(* POU TN_INPUT_CONTROL, ST *)
FUNCTION_BLOCK TN_INPUT_CONTROL
VAR_IN_OUT
	Xus_TN_SCREEN : us_TN_SCREEN;
	Xus_TN_INPUT_CONTROL : us_TN_INPUT_CONTROL;
END_VAR
VAR
	FB_TN_INPUT_SELECT_POPUP : TN_INPUT_SELECT_POPUP;
	FB_TN_INPUT_SELECT_TEXT : TN_INPUT_SELECT_TEXT;
	FB_TN_SC_WRITE_C : TN_SC_WRITE_C;
	FB_TN_INPUT_EDIT_LINE : TN_INPUT_EDIT_LINE;
END_VAR
VAR
	in_index : INT;
	in_Scroll_Offset : INT;
	in_Focus_new : INT;
	in_Focus_alt : INT;
	bo_Tool_Tip_Update : BOOL;
END_VAR

(*
version 1.0		10. mai 2010
programmer		ks
tested by		ks

TN_INPUT_CONTROL dient zur verwaltung und grafischen Darstellung der INPUT_CONTROL Elemente
*)
(* Bearbeitung freigegeben ? *)
IF (Xus_TN_INPUT_CONTROL.bo_Enable = FALSE) OR (Xus_TN_SCREEN.bo_Menue_Bar_Dialog = TRUE) THEN
	RETURN;
END_IF;

(* Fokus Reset durchführen *)
IF (Xus_TN_INPUT_CONTROL.bo_Reset_Fokus = TRUE) THEN
	Xus_TN_INPUT_CONTROL.bo_Reset_Fokus := FALSE;

	FOR in_index := INT#01 TO Xus_TN_INPUT_CONTROL.in_Count DO
		Xus_TN_INPUT_CONTROL.usa_TN_INPUT_CONTROL_DATA[in_index].bo_Focus := FALSE;
	END_FOR;

	IF (Xus_TN_INPUT_CONTROL.in_Count >= INT#01) THEN
		Xus_TN_INPUT_CONTROL.usa_TN_INPUT_CONTROL_DATA[1].bo_Focus := TRUE;
		Xus_TN_INPUT_CONTROL.in_Focus_at := INT#01;
	END_IF;

	Xus_TN_INPUT_CONTROL.bo_Update_all := TRUE;
END_IF;

IF (Xus_TN_SCREEN.bo_Modal_Dialog = FALSE) THEN
	(* TAB-Taste für Control-element wechsel auswerten *)
	IF (Xus_TN_SCREEN.by_Input_Exten_Code = BYTE#09) THEN

		in_Scroll_Offset := INT#01;

		(* Cursor-Oben Taste *)
	ELSIF (Xus_TN_SCREEN.by_Input_Exten_Code = BYTE#65) THEN

		in_Scroll_Offset := -1;

		(* Cursor-unten Taste *)
	ELSIF (Xus_TN_SCREEN.by_Input_Exten_Code = BYTE#66) THEN

		in_Scroll_Offset := INT#01;

	END_IF;
END_IF;

IF (in_Scroll_Offset <> INT#00) THEN  
	(* Grenzwerte überprüfen                                            *)

	Xus_TN_INPUT_CONTROL.in_Focus_at:=LIMIT(INT#01,Xus_TN_INPUT_CONTROL.in_Focus_at,Xus_TN_INPUT_CONTROL.in_Count);

	in_Focus_new := Xus_TN_INPUT_CONTROL.in_Focus_at + in_Scroll_Offset;

	IF (in_Focus_new > Xus_TN_INPUT_CONTROL.in_Count) THEN
		in_Focus_new := INT#1;
	END_IF;

	IF (in_Focus_new < INT#01) THEN
		in_Focus_new := Xus_TN_INPUT_CONTROL.in_Count;
	END_IF;

	in_Focus_alt := Xus_TN_INPUT_CONTROL.in_Focus_at;

	(* aktuellen Element den Fokus entziehen *)
	Xus_TN_INPUT_CONTROL.usa_TN_INPUT_CONTROL_DATA[in_Focus_alt].bo_Focus := FALSE;
	Xus_TN_INPUT_CONTROL.usa_TN_INPUT_CONTROL_DATA[in_Focus_alt].bo_Update_Input := TRUE;

	(* neuem Element den Fokus geben *)
	Xus_TN_INPUT_CONTROL.usa_TN_INPUT_CONTROL_DATA[in_Focus_new].bo_Focus  := TRUE;
	Xus_TN_INPUT_CONTROL.usa_TN_INPUT_CONTROL_DATA[in_Focus_new].bo_Update_Input := TRUE;

	Xus_TN_INPUT_CONTROL.in_Focus_at := in_Focus_new;

	bo_Tool_Tip_Update := TRUE;
	in_Scroll_Offset := INT#00;

END_IF;

(* Alle Elemente updaten ? *)
IF (Xus_TN_INPUT_CONTROL.bo_Update_all = TRUE) THEN
	FOR in_index := 1 TO Xus_TN_INPUT_CONTROL.in_Count DO
		Xus_TN_INPUT_CONTROL.usa_TN_INPUT_CONTROL_DATA[in_index].bo_Update_All := TRUE;
	END_FOR;
	Xus_TN_INPUT_CONTROL.bo_Update_all := FALSE;
	bo_Tool_Tip_Update := TRUE;
END_IF;

FOR in_index := 1 TO Xus_TN_INPUT_CONTROL.in_Count DO

	IF (Xus_TN_INPUT_CONTROL.usa_TN_INPUT_CONTROL_DATA[in_index].in_Type > INT#00) THEN

		IF (Xus_TN_INPUT_CONTROL.usa_TN_INPUT_CONTROL_DATA[in_index].bo_Focus = TRUE) THEN

			Xus_TN_INPUT_CONTROL.usa_TN_INPUT_CONTROL_DATA[in_index].by_Input_ASCII_Code  := Xus_TN_SCREEN.by_Input_ASCII_Code;
			Xus_TN_INPUT_CONTROL.usa_TN_INPUT_CONTROL_DATA[in_index].by_Input_Exten_Code  := Xus_TN_SCREEN.by_Input_Exten_Code;
			Xus_TN_INPUT_CONTROL.usa_TN_INPUT_CONTROL_DATA[in_index].bo_Input_ASCII_IsNum := Xus_TN_SCREEN.bo_Input_ASCII_IsNum;

			(* Tool-Tip Text ausgeben *)
			IF (bo_Tool_Tip_Update = TRUE) THEN

				FB_TN_SC_WRITE_C(	Iin_Y := Xus_TN_INPUT_CONTROL.in_ToolTip_Y,
									Iin_X := Xus_TN_INPUT_CONTROL.in_ToolTip_X,
									Iby_ATTR := Xus_TN_INPUT_CONTROL.by_ToolTip_Attr,
									Iin_OPTION := INT#02, (* Center-String *)
									Iin_LENGTH := Xus_TN_INPUT_CONTROL.in_ToolTip_Size,
									Ist_STRING := Xus_TN_INPUT_CONTROL.usa_TN_INPUT_CONTROL_DATA[in_index].st_Input_ToolTip,
									Xus_TN_SCREEN := Xus_TN_SCREEN);

				(* Flag rücksetzen *)
				bo_Tool_Tip_Update := FALSE;
			END_IF;
		END_IF;

		CASE Xus_TN_INPUT_CONTROL.usa_TN_INPUT_CONTROL_DATA[in_index].in_Type OF
		1:
			(* Edit-Line bearbeiten *)
			FB_TN_INPUT_EDIT_LINE(	Xus_TN_INPUT_CONTROL_DATA := Xus_TN_INPUT_CONTROL.usa_TN_INPUT_CONTROL_DATA[in_index],
									Xus_TN_SCREEN := Xus_TN_SCREEN);
		2:
			(* Select-Text bearbeiten *)
			FB_TN_INPUT_SELECT_TEXT(	Xus_TN_INPUT_CONTROL_DATA := Xus_TN_INPUT_CONTROL.usa_TN_INPUT_CONTROL_DATA[in_index],
										Xus_TN_SCREEN := Xus_TN_SCREEN);
		3:
			(* Select-Popup bearbeiten *)
			FB_TN_INPUT_SELECT_POPUP(	Xus_TN_INPUT_CONTROL_DATA := Xus_TN_INPUT_CONTROL.usa_TN_INPUT_CONTROL_DATA[in_index],
										Xus_TN_SCREEN := Xus_TN_SCREEN);
		END_CASE;

		IF (Xus_TN_INPUT_CONTROL.usa_TN_INPUT_CONTROL_DATA[in_index].bo_Focus = TRUE) THEN

			(* Cursor position von Element auf Screen übertragen *)
			Xus_TN_SCREEN.in_Cursor_X := Xus_TN_INPUT_CONTROL.usa_TN_INPUT_CONTROL_DATA[in_index].in_Cursor_X;
			Xus_TN_SCREEN.in_Cursor_Y := Xus_TN_INPUT_CONTROL.usa_TN_INPUT_CONTROL_DATA[in_index].in_Cursor_Y;

		END_IF;
	END_IF;
END_FOR;

(* revision history
ks	10. mai. 2010	rev 1.0
	original version
*)
END_FUNCTION_BLOCK

(* POU TN_INPUT_SELECT_POPUP, ST *)
FUNCTION_BLOCK TN_INPUT_SELECT_POPUP
VAR
	in_index : INT;
	in_Element_Count : INT;
	by_Cur_Key : BYTE;
	by_Attr : BYTE;
	st_String : STRING;
END_VAR
VAR
	us_TN_MENU_POPUP : us_TN_MENU_POPUP;
	FB_TN_INPUT_MENU_POPUP : TN_INPUT_MENU_POPUP;
	FB_TN_SC_WRITE : TN_SC_WRITE;
END_VAR
VAR_IN_OUT
	Xus_TN_SCREEN : us_TN_SCREEN;
	Xus_TN_INPUT_CONTROL_DATA : us_TN_INPUT_CONTROL_DATA;
END_VAR

(*
version 1.1		06. apr 2011
programmer		ks
tested by			ks

TN_SELECT_POPUP dient zur verwaltung und darstellung eines POPUP-Dialogs zur Elementeauswahl
*)
(* Benutzereingabe auswerten -> Selektion Text n *)
IF (Xus_TN_INPUT_CONTROL_DATA.bo_Focus = TRUE) THEN

	by_Cur_Key := Xus_TN_INPUT_CONTROL_DATA.by_Input_Exten_Code;

	IF (us_TN_MENU_POPUP.bo_Activ = FALSE) THEN
		us_TN_MENU_POPUP.by_Input_Exten_Code := BYTE#00;

		(* Return-Taste auswerten *)
		IF (by_Cur_Key = BYTE#13) THEN
			(* Popup-Menu parameter übergeben *)
			us_TN_MENU_POPUP.in_Y := Xus_TN_INPUT_CONTROL_DATA.in_Y;
			us_TN_MENU_POPUP.in_X := Xus_TN_INPUT_CONTROL_DATA.in_X;
			us_TN_MENU_POPUP.by_Attr_mF := Xus_TN_INPUT_CONTROL_DATA.by_Attr_mF;
			us_TN_MENU_POPUP.by_Attr_oF := Xus_TN_INPUT_CONTROL_DATA.by_Attr_oF;
			us_TN_MENU_POPUP.st_Menu_Text := Xus_TN_INPUT_CONTROL_DATA.st_Input_Data;
			us_TN_MENU_POPUP.bo_Create := TRUE;
			us_TN_MENU_POPUP.in_Cur_Item := INT#00;
		END_IF;

		IF (us_TN_MENU_POPUP.in_Cur_Item > INT#00) THEN
			Xus_TN_INPUT_CONTROL_DATA.in_selected := us_TN_MENU_POPUP.in_Cur_Item;
			Xus_TN_INPUT_CONTROL_DATA.bo_Input_Entered := TRUE;
			Xus_TN_INPUT_CONTROL_DATA.bo_Update_Input := TRUE;
			us_TN_MENU_POPUP.in_Cur_Item := INT#00;
		END_IF;

	ELSE
		us_TN_MENU_POPUP.by_Input_Exten_Code := by_Cur_Key;
	END_IF;

	(* Popup-Menu zyklisch aufrufen *)
	FB_TN_INPUT_MENU_POPUP(Xus_TN_MENU_POPUP := us_TN_MENU_POPUP, Xus_TN_SCREEN := Xus_TN_SCREEN);

END_IF;

(* Aktualisierung der Anzeige *)
IF (Xus_TN_INPUT_CONTROL_DATA.bo_Update_Input = TRUE) OR (Xus_TN_INPUT_CONTROL_DATA.bo_Update_All = TRUE) THEN

	(* Title-Text ausgeben *)
	IF Xus_TN_INPUT_CONTROL_DATA.bo_Update_All = TRUE THEN

		IF (Xus_TN_INPUT_CONTROL_DATA.in_Title_X_Offset = INT#00) AND (Xus_TN_INPUT_CONTROL_DATA.in_Title_Y_Offset = INT#00) THEN
			(* wenn Offset X,Y =0 dann Titlestring links vom Element positionieren *)
			FB_TN_SC_WRITE.Iin_Y := Xus_TN_INPUT_CONTROL_DATA.in_Y;
			FB_TN_SC_WRITE.Iin_X := Xus_TN_INPUT_CONTROL_DATA.in_X - LEN(Xus_TN_INPUT_CONTROL_DATA.st_Title_String);

		ELSE
			(* Title-Text durch Row, Color-Offset ausgeben *)
			FB_TN_SC_WRITE.Iin_Y := Xus_TN_INPUT_CONTROL_DATA.in_Y + Xus_TN_INPUT_CONTROL_DATA.in_Title_Y_Offset;
			FB_TN_SC_WRITE.Iin_X := Xus_TN_INPUT_CONTROL_DATA.in_X + Xus_TN_INPUT_CONTROL_DATA.in_Title_X_Offset;
		END_IF;

		(* Title-Text durch Row, Color-Offset ausgeben *)
		FB_TN_SC_WRITE(	Iby_ATTR := Xus_TN_INPUT_CONTROL_DATA.by_Title_Attr,
						Ist_STRING := Xus_TN_INPUT_CONTROL_DATA.st_Title_String,
						Xus_TN_SCREEN := Xus_TN_SCREEN);
	END_IF;

	in_Element_Count := ELEMENT_COUNT(SEP:=BYTE#35,ELEMENT:=Xus_TN_INPUT_CONTROL_DATA.st_Input_Data);

	IF in_Element_Count > INT#00 THEN

		Xus_TN_INPUT_CONTROL_DATA.in_selected:=LIMIT(1,Xus_TN_INPUT_CONTROL_DATA.in_selected,in_Element_Count);

		in_index := Xus_TN_INPUT_CONTROL_DATA.in_selected;

		st_String := ELEMENT_GET(SEP:=BYTE#35,POS:=in_index - 1,ELEMENT:=Xus_TN_INPUT_CONTROL_DATA.st_Input_Data);

		st_String:= FIX(str:=st_String,
						L:=LEN(Xus_TN_INPUT_CONTROL_DATA.st_Input_Mask),
						C:=BYTE#32,
						M:=Xus_TN_INPUT_CONTROL_DATA.in_Input_Option);


		Xus_TN_INPUT_CONTROL_DATA.st_Input_String := st_String;

		IF Xus_TN_INPUT_CONTROL_DATA.bo_Focus = TRUE THEN
			by_Attr := Xus_TN_INPUT_CONTROL_DATA.by_Attr_mF;
		ELSE
			by_Attr := Xus_TN_INPUT_CONTROL_DATA.by_Attr_oF;
		END_IF;

		FB_TN_SC_WRITE(	Iin_X := Xus_TN_INPUT_CONTROL_DATA.in_X,
								Iin_Y := Xus_TN_INPUT_CONTROL_DATA.in_Y,
								Iby_ATTR := by_Attr,
								Ist_STRING := st_String,
								Xus_TN_SCREEN := Xus_TN_SCREEN );
	END_IF;

	(* Cursor auf aktuelle Position setzen *)
	Xus_TN_INPUT_CONTROL_DATA.in_Cursor_X := Xus_TN_INPUT_CONTROL_DATA.in_X;
	Xus_TN_INPUT_CONTROL_DATA.in_Cursor_Y := Xus_TN_INPUT_CONTROL_DATA.in_Y;

	(* Update-Flag's rücksetzen *)
	Xus_TN_INPUT_CONTROL_DATA.bo_Update_All   := FALSE;
	Xus_TN_INPUT_CONTROL_DATA.bo_Update_Input := FALSE;

END_IF;

(* revision history

ks	06. apr. 2011	rev 1.1
	list_len und list_get durch element_count und element_get ersetzt

ks	10. mai. 2010	rev 1.0
	original version
*)
END_FUNCTION_BLOCK

(* POU TN_INPUT_MENU_POPUP, ST *)
FUNCTION_BLOCK TN_INPUT_MENU_POPUP
VAR
	FB_TN_SC_AREA_SAVE : TN_SC_AREA_SAVE;
	FB_TN_SC_AREA_RESTORE : TN_SC_AREA_RESTORE;
	FB_TN_SC_LINE : TN_SC_LINE;
	FB_TN_SC_ADD_SHADOW : TN_SC_ADD_SHADOW;
	FB_TN_SC_BOX : TN_SC_BOX;
	FB_TN_SC_WRITE_C : TN_SC_WRITE_C;
END_VAR
VAR
	in_ROW : INT;
	in_ROWS : INT;
	in_COL : INT;
	in_COLS : INT;
	in_index : INT;
	in_Count : INT;
	in_Scroll_Offset : INT;
	by_ATTR : BYTE;
END_VAR
VAR_IN_OUT
	Xus_TN_MENU_POPUP : us_TN_MENU_POPUP;
	Xus_TN_SCREEN : us_TN_SCREEN;
END_VAR

(*
version 1.1		06. apr 2011
programmer		ks
tested by			ks

TN_MENU_POPUP dient zur verwaltung und darstellung eines MENU-POPUP
*)
(* sicherstellen das rechteck immer innerhalb screen positioniert wird *)

IF (Xus_TN_MENU_POPUP.bo_Activ = FALSE) AND (Xus_TN_MENU_POPUP.bo_Create = TRUE) THEN
	Xus_TN_MENU_POPUP.bo_Activ := TRUE;
	Xus_TN_MENU_POPUP.bo_Create := FALSE;
	Xus_TN_MENU_POPUP.bo_Destroy := FALSE;
	Xus_TN_MENU_POPUP.bo_Update := TRUE;

  (* Sub-Menu-Texte *)

	Xus_TN_MENU_POPUP.in_Menu_E_Count := ELEMENT_COUNT(SEP:=BYTE#35,ELEMENT:=Xus_TN_MENU_POPUP.st_Menu_Text);

	(* Anzahl Zeilen (Sub-Menu-Texte) bestimmen *)
	Xus_TN_MENU_POPUP.in_Rows := Xus_TN_MENU_POPUP.in_Menu_E_Count;

	(* längsten Sub-Menu-Text suchen *)
	Xus_TN_MENU_POPUP.in_Cols := INT#00;

	FOR in_Count := INT#01 TO Xus_TN_MENU_POPUP.in_Rows DO;
		Xus_TN_MENU_POPUP.in_Cols:=MAX(LEN(ELEMENT_GET(SEP:=BYTE#35,POS:=in_Count - 1,ELEMENT:=Xus_TN_MENU_POPUP.st_Menu_Text)),Xus_TN_MENU_POPUP.in_Cols);
	END_FOR;

	(* Horizontale Position überprüfen und korrigieren *)
	IF (Xus_TN_MENU_POPUP.in_X + Xus_TN_MENU_POPUP.in_Cols) > INT#75 THEN
		Xus_TN_MENU_POPUP.in_X := INT#79 - Xus_TN_MENU_POPUP.in_Cols - INT#04;
	END_IF;

  (* Vertikale Position überprüfen und korrigieren *)
	IF (Xus_TN_MENU_POPUP.in_Y + Xus_TN_MENU_POPUP.in_ROWS) > INT#21 THEN
		Xus_TN_MENU_POPUP.in_Y := INT#23 - Xus_TN_MENU_POPUP.in_ROWS - INT#2;
	END_IF;

	Xus_TN_SCREEN.bo_Modal_Dialog := TRUE;

	(* Hintergrund sichern *)
	FB_TN_SC_AREA_SAVE(	Iin_X1 := Xus_TN_MENU_POPUP.in_X,
									Iin_Y1 := Xus_TN_MENU_POPUP.in_Y,
									Iin_X2 := Xus_TN_MENU_POPUP.in_X + Xus_TN_MENU_POPUP.in_Cols + INT#04,
									Iin_Y2 := Xus_TN_MENU_POPUP.in_Y + Xus_TN_MENU_POPUP.in_Rows + INT#02,
									Xus_TN_SCREEN := Xus_TN_SCREEN);

	(* Rahmen für Submenu zeichnen *)
	FB_TN_SC_BOX(	Iin_X1 := Xus_TN_MENU_POPUP.in_X,
					Iin_Y1 := Xus_TN_MENU_POPUP.in_Y,
					Iin_X2 := Xus_TN_MENU_POPUP.in_X + Xus_TN_MENU_POPUP.in_Cols + INT#03,
					Iin_Y2 := Xus_TN_MENU_POPUP.in_Y + Xus_TN_MENU_POPUP.in_Rows + INT#01,
					Iby_FILL := BYTE#32, (* Füllung *)
					Iin_BORDER := INT#01, (* Single-Line Border *)
					Iby_ATTR := Xus_TN_MENU_POPUP.by_Attr_oF,
					Xus_TN_SCREEN := Xus_TN_SCREEN);

	(* Shadow für Submenu zeichnen *)
	FB_TN_SC_ADD_SHADOW(Iin_X1 := Xus_TN_MENU_POPUP.in_X + INT#1,
						Iin_Y1 := Xus_TN_MENU_POPUP.in_Y + INT#1,
						Iin_X2 := Xus_TN_MENU_POPUP.in_X + Xus_TN_MENU_POPUP.in_Cols + INT#04,
						Iin_Y2 := Xus_TN_MENU_POPUP.in_Y + Xus_TN_MENU_POPUP.in_Rows + INT#02,
						Iin_OPTION := INT#00,
						Xus_TN_SCREEN := Xus_TN_SCREEN);

	(* Parameter laden *)
	in_COL := Xus_TN_MENU_POPUP.in_X;
	in_ROW := Xus_TN_MENU_POPUP.in_Y;
	in_ROWS := Xus_TN_MENU_POPUP.in_Rows;
	in_COLS := Xus_TN_MENU_POPUP.in_Cols;

	(* Trennlinien zeichnen *)
	in_COLS := in_COLS + INT#02; (* Text um 2 Zeichen verlängern *)

	FOR in_Count := INT#01 TO Xus_TN_MENU_POPUP.in_Menu_E_Count DO;
		in_ROW := in_ROW + INT#01;

		IF ELEMENT_GET(SEP:=BYTE#35,POS:=in_Count - 1,ELEMENT:=Xus_TN_MENU_POPUP.st_Menu_Text) = '-' THEN

			FB_TN_SC_LINE(	Iin_Y1 := in_ROW,
							Iin_X1 := in_COL,
							Iin_Y2 := in_ROW,
							Iin_X2 := in_COL + in_COLS + INT#01,
							Iby_ATTR := Xus_TN_MENU_POPUP.by_Attr_oF,
							Iby_BORDER := BYTE#01,
							Xus_TN_SCREEN := Xus_TN_SCREEN);
		END_IF;
	END_FOR;
END_IF;

IF (Xus_TN_MENU_POPUP.bo_Activ = TRUE) THEN

	CASE BYTE_TO_INT(Xus_TN_MENU_POPUP.by_Input_Exten_Code) OF

	65: (* Cursor oben *)
		in_Scroll_Offset := -1;
		Xus_TN_MENU_POPUP.bo_Update := TRUE;

	66: (* Cursor unten *)
		in_Scroll_Offset := 1;
		Xus_TN_MENU_POPUP.bo_Update := TRUE;

	13:  (* Enter *)
		Xus_TN_MENU_POPUP.bo_Destroy := TRUE;

	27:  (* Escape*)
		Xus_TN_MENU_POPUP.bo_Destroy := TRUE;
		Xus_TN_MENU_POPUP.in_Cur_Item := INT#00;

	67..68: (* Cursor links oder rechts *)
		Xus_TN_MENU_POPUP.bo_Destroy := TRUE;
		Xus_TN_MENU_POPUP.in_Cur_Item := INT#00;

	END_CASE;
END_IF;

(* POPUP-Menu updaten *)
IF (Xus_TN_MENU_POPUP.bo_Activ = TRUE) AND (Xus_TN_MENU_POPUP.bo_Update = TRUE) THEN

	Xus_TN_MENU_POPUP.bo_Update := FALSE;

	(* überprüfung + nächstes anwählbares Sub-Menu suchen *)
	in_index := Xus_TN_MENU_POPUP.in_Cur_Item;

	IF (in_index < INT#01) OR (in_index > Xus_TN_MENU_POPUP.in_Menu_E_Count) THEN
		in_Scroll_Offset := INT#01;
		in_index := Xus_TN_MENU_POPUP.in_Menu_E_Count;
	END_IF;

	(* aktueller Index steht auf Trennzeichen -> ändern *)
	IF ELEMENT_GET(SEP:=BYTE#35,POS:=in_index-1,ELEMENT:=Xus_TN_MENU_POPUP.st_Menu_Text) = '-' THEN
		in_Scroll_Offset := INT#01;
	END_IF;

	(* Scroll-Offset *)
	IF in_Scroll_Offset <> INT#00 THEN

		FOR in_Count := INT#01 TO Xus_TN_MENU_POPUP.in_Menu_E_Count DO;

			in_index:=INC2(in_index,in_Scroll_Offset,1,Xus_TN_MENU_POPUP.in_Menu_E_Count);

			IF ELEMENT_GET(SEP:=BYTE#35,POS:=in_index - 1,ELEMENT:=Xus_TN_MENU_POPUP.st_Menu_Text) <> '-' THEN
				EXIT;
			END_IF;

		END_FOR;
	END_IF;

	Xus_TN_MENU_POPUP.in_Cur_Item := in_index;
	in_Scroll_Offset := INT#00;

	(* Parameter laden *)
	in_COL  := Xus_TN_MENU_POPUP.in_X;
	in_ROW  := Xus_TN_MENU_POPUP.in_Y;
	in_ROWS := Xus_TN_MENU_POPUP.in_Rows;
	in_COLS := Xus_TN_MENU_POPUP.in_Cols;

	(* SUB-MENU-Titel ausgeben *)
	in_COLS := in_COLS + INT#02; (* Text um 2 Zeichen verlängern *)

	FOR in_Count := INT#01 TO Xus_TN_MENU_POPUP.in_Menu_E_Count DO;

		in_ROW := in_ROW + INT#01;

		(* Zeichenfarbe bestimmen *)
		IF in_Count = Xus_TN_MENU_POPUP.in_Cur_Item THEN
			by_ATTR := Xus_TN_MENU_POPUP.by_Attr_mF;
		ELSE
			by_ATTR := Xus_TN_MENU_POPUP.by_Attr_oF;
		END_IF;

		FB_TN_SC_WRITE_C.Ist_STRING := ELEMENT_GET(SEP:=BYTE#35,POS:=in_Count - 1,ELEMENT:=Xus_TN_MENU_POPUP.st_Menu_Text);

		IF FB_TN_SC_WRITE_C.Ist_STRING <> '-' THEN

			FB_TN_SC_WRITE_C(	Iin_Y := in_ROW,
								Iin_X := in_COL + INT#01,
								Iby_ATTR := by_ATTR,
								Iin_LENGTH := in_COLS,
								Iin_OPTION := INT#02, (* Center *)
								Xus_TN_SCREEN := Xus_TN_SCREEN);
		END_IF;
	END_FOR;
END_IF;

(* POPUP-Menu entfernen (Destroy) *)
IF (Xus_TN_MENU_POPUP.bo_Activ = TRUE) AND (Xus_TN_MENU_POPUP.bo_Destroy = TRUE) THEN

	Xus_TN_MENU_POPUP.bo_Destroy := FALSE;
	Xus_TN_MENU_POPUP.bo_Activ := FALSE;

	(* alten Hintergrund aus Speicher wiederherstellen *)
	FB_TN_SC_AREA_RESTORE(Xus_TN_SCREEN := Xus_TN_SCREEN);

	Xus_TN_SCREEN.bo_Modal_Dialog := FALSE;
END_IF;

(* revision history

ks	06. apr. 2011	rev 1.1
	list_len und list_get durch element_count und element_get ersetzt

ks	10. mai. 2010	rev 1.0
	original version
*)
END_FUNCTION_BLOCK

(* POU TN_SC_AREA_SAVE, ST *)
FUNCTION_BLOCK TN_SC_AREA_SAVE
VAR
	in_Offset_1 : INT;
	in_Offset_2 : INT;
	in_Y : INT;
	in_X : INT;
END_VAR
VAR_INPUT
	Iin_Y1 : INT;
	Iin_X1 : INT;
	Iin_Y2 : INT;
	Iin_X2 : INT;
END_VAR
VAR_IN_OUT
	Xus_TN_SCREEN : us_TN_SCREEN;
END_VAR

(*
version 1.0		10. mai 2010
programmer		ks
tested by		ks

TN_SC_AREA_SAVE sichert den angegebenen Bildschirmbereich in einem Buffer
*)
IF TN_SC_XY2_ERROR(Iin_X1,Iin_Y1,Iin_X2,Iin_Y2) THEN RETURN; END_IF;

(* Parameter ablegen *)
Xus_TN_SCREEN.bya_BACKUP[0] := BYTE#1;
Xus_TN_SCREEN.bya_BACKUP[1] := INT_TO_BYTE(Iin_X1);
Xus_TN_SCREEN.bya_BACKUP[2] := INT_TO_BYTE(Iin_Y1); 
Xus_TN_SCREEN.bya_BACKUP[3] := INT_TO_BYTE(Iin_X2);
Xus_TN_SCREEN.bya_BACKUP[4] := INT_TO_BYTE(Iin_Y2);

in_Offset_2 := 5;
(* CHAR und COLOR in BUFFER sichern *)
FOR in_Y := Iin_Y1 TO Iin_Y2 DO

	in_Offset_1 := (in_Y * 80) + Iin_X1;
	FOR in_X := Iin_X1 TO Iin_X2 DO
		Xus_TN_SCREEN.bya_BACKUP[in_Offset_2] := Xus_TN_SCREEN.bya_CHAR[in_Offset_1];
		in_Offset_2 := in_Offset_2 + INT#01;
		Xus_TN_SCREEN.bya_BACKUP[in_Offset_2] := Xus_TN_SCREEN.bya_COLOR[in_Offset_1];
		in_Offset_2 := in_Offset_2 + INT#01;
		in_Offset_1 := in_Offset_1 + INT#01;
	END_FOR;
END_FOR;

(* revision history
ks	10. mai. 2010	rev 1.0
	original version
*)
END_FUNCTION_BLOCK

(* POU TN_SC_XY2_ERROR, ST *)
FUNCTION TN_SC_XY2_ERROR : BOOL
VAR_INPUT
	X1 : INT;
	Y1 : INT;
	X2 : INT;
	Y2 : INT;
END_VAR

(*
version 1.0		10. mai 2010
programmer		ks
tested by		ks

TN_SC_XY2_ERROR prüft ob die angegenene Koordinaten die einen rechteckigen Bereich angeben gültig sind 
*)
(* min und max werte prüfen *)
TN_SC_XY2_ERROR := Y1 < 0 OR X1 < 0 OR Y2 < 0 OR X2 < 0 OR Y1 > 23 OR X1 > 79 OR Y2 > 23 OR X2 > 79;

(* revision history
ks	10. mai. 2010	rev 1.0
	original version
*)
END_FUNCTION

(* POU TN_SC_AREA_RESTORE, ST *)
FUNCTION_BLOCK TN_SC_AREA_RESTORE
VAR
	in_Offset_1 : INT;
	in_Offset_2 : INT;
	in_Y : INT;
	in_X : INT;
	in_Y1 : INT;
	in_X1 : INT;
	in_Y2 : INT;
	in_X2 : INT;
END_VAR
VAR_IN_OUT
	Xus_TN_SCREEN : us_TN_SCREEN;
END_VAR

(*
version 1.0		10. mai 2010
programmer		ks
tested by		ks

TN_SC_AREA_RESTORE stellt den zuvor gesicherten Bildschirmbereich wieder her
*)
IF Xus_TN_SCREEN.bya_BACKUP[0] > BYTE#00 THEN

	(* Parameter auslesen *)
	in_X1 := BYTE_TO_INT(Xus_TN_SCREEN.bya_BACKUP[1]);
	in_Y1 := BYTE_TO_INT(Xus_TN_SCREEN.bya_BACKUP[2]);
	in_X2 := BYTE_TO_INT(Xus_TN_SCREEN.bya_BACKUP[3]);
	in_Y2 := BYTE_TO_INT(Xus_TN_SCREEN.bya_BACKUP[4]);

	IF TN_SC_XY2_ERROR(in_X1,in_Y1,in_X2,in_Y2) THEN RETURN; END_IF;
	in_Offset_2 := 5;

	(* CHAR und COLOR von BUFFER wiederherstellen *)
	FOR in_Y := in_Y1 TO in_Y2 DO

		Xus_TN_SCREEN.bya_Line_Update[in_Y] := TRUE; (* Zeile zum Updaten freigeben *)
		in_Offset_1 := (in_Y * 80) + in_X1;

		FOR in_X := in_X1 TO in_X2 DO

			Xus_TN_SCREEN.bya_CHAR[in_Offset_1] := Xus_TN_SCREEN.bya_BACKUP[in_Offset_2];
			in_Offset_2 := in_Offset_2 + INT#01;

			Xus_TN_SCREEN.bya_COLOR[in_Offset_1] := Xus_TN_SCREEN.bya_BACKUP[in_Offset_2];
			in_Offset_2 := in_Offset_2 + INT#01;
			in_Offset_1 := in_Offset_1 + INT#01;

		END_FOR;
	END_FOR;

	(* Daten als ungültig markieren *)
	Xus_TN_SCREEN.bya_BACKUP[0] := BYTE#00;
END_IF;

(* revision history
ks	10. mai. 2010	rev 1.0
	original version
*)
END_FUNCTION_BLOCK

(* POU TN_SC_LINE, ST *)
FUNCTION_BLOCK TN_SC_LINE
VAR
	by_Connect_Left_Char : BYTE;
	by_Connect_Right_Char : BYTE;
	by_Connect_Top_Char : BYTE;
	by_Connect_Bottom_Char : BYTE;
	by_Connect_Cruz_Char : BYTE;
	by_Vertikal_Line_Char : BYTE;
	by_Horzontal_Line_Char : BYTE;
	by_old_Char : BYTE;
	in_Offset_1 : INT;
	in_ROW_Index : INT;
	in_COL_Index : INT;
	by_Char : BYTE;
END_VAR
VAR_INPUT
	Iin_X1 : INT;
	Iin_Y1 : INT;
	Iin_X2 : INT;
	Iin_Y2 : INT;
	Iby_ATTR : BYTE;
	Iby_BORDER : BYTE;
END_VAR
VAR_IN_OUT
	Xus_TN_SCREEN : us_TN_SCREEN;
END_VAR

(*
version 1.0		10. mai 2010
programmer		ks
tested by		ks

TN_SC_LINE zeichnet horizontale und vertikale Linien
*)
IF TN_SC_XY2_ERROR(Iin_X1,Iin_Y1,Iin_X2,Iin_Y2) THEN RETURN; END_IF;

(* Bordertype bestimmen *)
IF Iby_Border = BYTE#01 THEN (* Single Line *)
	by_Connect_Top_Char := BYTE#16#C2;
	by_Connect_Bottom_Char := BYTE#16#C1;
	by_Connect_Left_Char := BYTE#16#C3;
	by_Connect_Right_Char := BYTE#16#B4;
	by_Horzontal_Line_Char := BYTE#16#C4;
	by_Vertikal_Line_Char := BYTE#16#B3;
	by_Connect_Cruz_Char := BYTE#16#C5;
ELSIF Iby_Border = BYTE#02 THEN	(* Double Linie *)
	by_Connect_Top_Char := BYTE#16#CB;
	by_Connect_Bottom_Char := BYTE#16#CA;
	by_Connect_Left_Char := BYTE#16#CC;
	by_Connect_Right_Char := BYTE#16#B9;
	by_Horzontal_Line_Char := BYTE#16#CD;
	by_Vertikal_Line_Char := BYTE#16#BA;
	by_Connect_Cruz_Char := BYTE#16#CE;
ELSE (* Full Linie *)
	by_Connect_Top_Char := Iby_Border;
	by_Connect_Bottom_Char := Iby_Border;
	by_Connect_Left_Char := Iby_Border;
	by_Connect_Right_Char := Iby_Border;
	by_Horzontal_Line_Char := Iby_Border;
	by_Vertikal_Line_Char := Iby_Border;
	by_Connect_Cruz_Char := Iby_Border;
END_IF;

(* Vertikale Linie zeichnen *)
IF Iin_X1 = Iin_X2 THEN
	in_Offset_1 := (Iin_Y1 * 80) + Iin_X1;
	FOR in_ROW_Index := Iin_Y1 TO Iin_Y2 DO
		by_old_Char := Xus_TN_SCREEN.bya_CHAR[in_Offset_1]; (* bestehendes Zeichen auslesen *)
		by_Char := by_Vertikal_Line_Char; (* Standardzeichen vorbelegen *)
		IF by_old_Char = by_Horzontal_Line_Char THEN (* Schnittpunkt erkannt *)
			IF in_ROW_Index = Iin_Y1 THEN (* Anfang der Linie behandeln *)
				by_Char := by_Connect_Top_Char;
			ELSIF in_ROW_Index = Iin_Y2 THEN (* Ende der Linie behandeln *)
				by_Char := by_Connect_Bottom_Char;
			ELSE (* Kreuzungspunkt behandeln *)
				by_Char := by_Connect_Cruz_Char;
			END_IF;
		END_IF;
		Xus_TN_SCREEN.bya_Line_Update[in_ROW_Index] := TRUE; (* Zeile zum Updaten freigeben *)
		Xus_TN_SCREEN.bya_CHAR[in_Offset_1] := by_Char;
		Xus_TN_SCREEN.bya_COLOR[in_Offset_1] := Iby_Attr;
		in_Offset_1 := in_Offset_1 + 80;
	END_FOR;

ELSIF Iin_Y1 = Iin_Y2 THEN (* Horzontale Linie zeichnen *)
	Xus_TN_SCREEN.bya_Line_Update[Iin_Y1] := TRUE; (* Zeile zum Updaten freigeben *)
	in_Offset_1 := (Iin_Y1 * 80) + Iin_X1;
	FOR in_COL_Index := Iin_X1 TO Iin_X2 DO
		by_old_Char := Xus_TN_SCREEN.bya_CHAR[in_Offset_1]; (* bestehendes Zeichen auslesen *)
		by_Char := by_Horzontal_Line_Char; (* Standardzeichen vorbelegen *)
		IF by_old_Char = by_Vertikal_Line_Char THEN (* Schnittpunkt erkannt *)
			IF in_COL_Index = Iin_X1 THEN (* Anfang der Linie behandeln *)
				by_Char := by_Connect_Left_Char;
			ELSIF in_COL_Index = Iin_X2 THEN (* Ende der Linie behandeln *)
				by_Char := by_Connect_Right_Char;
			ELSE (* Kreuzungspunkt behandeln *)
				by_Char := by_Connect_Cruz_Char;
			END_IF;
		END_IF;
		Xus_TN_SCREEN.bya_CHAR[in_Offset_1] := by_Char;
		Xus_TN_SCREEN.bya_COLOR[in_Offset_1] := Iby_Attr;
		in_Offset_1 := in_Offset_1 + 1;
	END_FOR;
END_IF;

(* revision history
ks	10. mai. 2010	rev 1.0
	original version
*)
END_FUNCTION_BLOCK

(* POU TN_SC_ADD_SHADOW, ST *)
FUNCTION_BLOCK TN_SC_ADD_SHADOW
VAR
	in_Offset : INT;
	in_X : INT;
	in_Y : INT;
END_VAR
VAR_INPUT
	Iin_Y1 : INT;
	Iin_X1 : INT;
	Iin_Y2 : INT;
	Iin_X2 : INT;
	Iin_OPTION : INT;
END_VAR
VAR_IN_OUT
	Xus_TN_SCREEN : us_TN_SCREEN;
END_VAR

(*
version 1.0		10. mai 2010
programmer		ks
tested by		ks

TN_SC_ADD_SHADOW zeichnet auf der linken und unteren Seite eines rechteckigen Bereiches einen Schatten
*)
IF TN_SC_XY2_ERROR(Iin_X1,Iin_Y1,Iin_X2,Iin_Y2) THEN RETURN; END_IF;

IF Iin_Y1 < 0 OR Iin_X1 < 0 OR Iin_Y2 < 0 OR Iin_X2 < 0 THEN RETURN; END_IF; (* min werte prüfen *)
IF Iin_Y1 > 23 OR Iin_X1 > 79 OR Iin_Y2 > 23 OR Iin_X2 > 79 THEN RETURN; END_IF; (* max werte prüfen *)

in_Offset := (Iin_Y1 * 80) + Iin_X2;

IF Iin_OPTION = INT#00 THEN
	(* Schatten durch Farbanpassung erzeugen *)
	FOR in_Y := Iin_Y1 TO Iin_Y2 DO
		Xus_TN_SCREEN.bya_COLOR[in_Offset] := TN_SC_SHADOW_ATTR(Xus_TN_SCREEN.bya_COLOR[in_Offset]);
		in_Offset := in_Offset + 80;
		Xus_TN_SCREEN.bya_Line_Update[in_Y] := TRUE; (* Zeile für Update eintragen *)
	END_FOR;
ELSE
	(* Schatten durch Farbe Schwarz und Leerzeichen erzeugen *)
	FOR in_Y := Iin_Y1 TO Iin_Y2 DO
		Xus_TN_SCREEN.bya_COLOR[in_Offset] := BYTE#00;
		Xus_TN_SCREEN.bya_CHAR[in_Offset] := BYTE#32;
		in_Offset := in_Offset + 80;
		Xus_TN_SCREEN.bya_Line_Update[in_Y] := TRUE; (* Zeile für Update eintragen *)
	END_FOR;
END_IF;

in_Offset := (Iin_Y2 * 80) + Iin_X1;

IF Iin_OPTION = INT#00 THEN
	(* Schatten durch Farbanpassung erzeugen *)
	FOR in_X  := Iin_X1 TO Iin_X2 DO
		Xus_TN_SCREEN.bya_COLOR[in_Offset] := TN_SC_SHADOW_ATTR(Xus_TN_SCREEN.bya_COLOR[in_Offset]);
		in_Offset := in_Offset + 1;
	END_FOR;
ELSE
	(* Schatten durch Farbe Schwarz und Leerzeichen erzeugen *)
	FOR in_X  := Iin_X1 TO Iin_X2 DO
		Xus_TN_SCREEN.bya_COLOR[in_Offset] := BYTE#00;
		Xus_TN_SCREEN.bya_CHAR[in_Offset] := BYTE#32;
		in_Offset := in_Offset + 1;
	END_FOR;
END_IF;

(* revision history
ks	10. mai. 2010	rev 1.0
	original version
*)
END_FUNCTION_BLOCK

(* POU TN_SC_SHADOW_ATTR, ST *)
FUNCTION TN_SC_SHADOW_ATTR : BYTE
VAR_INPUT
	Iby_ATTR : BYTE;
END_VAR

(*
version 1.0		10. mai 2010
programmer		ks
tested by		ks

TN_SC_SHADOW_ATTR berechnet aus einem normalen einem abgedunkelten Farbcode
*)
(* Background Farbe auf Schwarz ändern      *)
(* und dunkle Fordergrundfarben einschalten *)  
TN_SC_SHADOW_ATTR := ((Iby_ATTR AND BYTE#2#11110000) OR BYTE#2#00001000);

(* revision history
ks	10. mai. 2010	rev 1.0
	original version
*)
END_FUNCTION

(* POU TN_SC_BOX, ST *)
FUNCTION_BLOCK TN_SC_BOX
VAR
	FB_TN_SC_FILL : TN_SC_FILL;
	by_BorderChar_L_T : BYTE;
	by_BorderChar_T : BYTE;
	by_BorderChar_B : BYTE;
	by_BorderChar_R_T : BYTE;
	by_BorderChar_L : BYTE;
	by_BorderChar_R : BYTE;
	by_BorderChar_L_B : BYTE;
	by_BorderChar_R_B : BYTE;
	in_Y : INT;
	in_X : INT;
	in_Border_Offset : INT;
	in_Offset_1 : INT;
	in_Offset_2 : INT;
END_VAR
VAR_INPUT
	Iin_Y1 : INT;
	Iin_X1 : INT;
	Iin_Y2 : INT;
	Iin_X2 : INT;
	Iby_FILL : BYTE;
	Iby_ATTR : BYTE;
	Iin_BORDER : INT;
END_VAR
VAR_IN_OUT
	Xus_TN_SCREEN : us_TN_SCREEN;
END_VAR

(*
version 1.0		10. mai 2010
programmer		ks
tested by		ks

TN_SC_BOX füllt einen rechteckigen Bereich mit einem Zeichen und zeichnet eine Umrandung
*)
IF TN_SC_XY2_ERROR(Iin_X1,Iin_Y1,Iin_X2,Iin_Y2) THEN RETURN; END_IF;

(* Bordertype bestimmen *)
CASE Iin_Border OF
0:
	in_Border_Offset := 0;
1:
	by_BorderChar_L_T := BYTE#218; (* links oben *)
	by_BorderChar_T := BYTE#196; (* oben *)
	by_BorderChar_R_T := BYTE#191; (* rechts oben *)
	by_BorderChar_L := BYTE#179; (* links *)
	by_BorderChar_R := BYTE#179; (* rechts *)
	by_BorderChar_B := BYTE#196; (* unten *)
	by_BorderChar_L_B := BYTE#217; (* links unten *)
	by_BorderChar_R_B := BYTE#192; (* rechts unten *)
	in_Border_Offset := 1;
 2:
	by_BorderChar_L_T := BYTE#201;
	by_BorderChar_T := BYTE#205;
	by_BorderChar_R_T := BYTE#187;
	by_BorderChar_L := BYTE#186;
	by_BorderChar_R := BYTE#186;
	by_BorderChar_B := BYTE#205;
	by_BorderChar_L_B := BYTE#188;
	by_BorderChar_R_B := BYTE#200;
	in_Border_Offset := 1;
ELSE
	by_BorderChar_L_T := BYTE#32;
	by_BorderChar_T := BYTE#32;
	by_BorderChar_R_T := BYTE#32;
	by_BorderChar_L := BYTE#32;
	by_BorderChar_R := BYTE#32;
	by_BorderChar_B := BYTE#32;
	by_BorderChar_L_B := BYTE#32;
	by_BorderChar_R_B := BYTE#32;
	in_Border_Offset := 1;

END_CASE;

IF Iby_FILL > BYTE#0 THEN (* FILL Zeichen vorhanden ? -> Box zeichnen *)

	(* Fill-Function um eine Zeichenreihe kleiner zeichnen *)
	FB_TN_SC_FILL(	Iin_Y1 := Iin_Y1 + in_Border_Offset,
					Iin_X1 := Iin_X1 + in_Border_Offset,
					Iin_Y2 := Iin_Y2 - in_Border_Offset,
					Iin_X2 := Iin_X2 - in_Border_Offset,
					Iby_CHAR := Iby_FILL,
					Iby_Attr := Iby_ATTR,
					Xus_TN_SCREEN := Xus_TN_SCREEN);
END_IF;

IF Iin_BORDER = 0 THEN RETURN; END_IF;

(* linken und rechten Rand ausgeben *)

in_Offset_1 := (Iin_Y1 * 80) + Iin_X1;
in_Offset_2 := (Iin_Y1 * 80) + Iin_X2;

FOR in_Y := Iin_Y1 TO Iin_Y2 DO

	(* Zeile zum Updaten freigeben *)
	Xus_TN_SCREEN.bya_Line_Update[in_Y] := TRUE;

	Xus_TN_SCREEN.bya_CHAR[in_Offset_1] := by_BorderChar_L;
	Xus_TN_SCREEN.bya_COLOR[in_Offset_1] := Iby_Attr;

	Xus_TN_SCREEN.bya_CHAR[in_Offset_2] := by_BorderChar_R;
	Xus_TN_SCREEN.bya_COLOR[in_Offset_2] := Iby_Attr;

	in_Offset_1 := in_Offset_1 + 80;
	in_Offset_2 := in_Offset_2 + 80;

END_FOR;

(* unteren und oberen Rand ausgeben *)
in_Offset_1 := (Iin_Y1 * 80) + Iin_X1;
in_Offset_2 := (Iin_Y2 * 80) + Iin_X1;

FOR in_X := Iin_X1 TO Iin_X2 DO

	Xus_TN_SCREEN.bya_CHAR[in_Offset_1] := by_BorderChar_T;
	Xus_TN_SCREEN.bya_COLOR[in_Offset_1] := Iby_Attr;

	Xus_TN_SCREEN.bya_CHAR[in_Offset_2] := by_BorderChar_B;
	Xus_TN_SCREEN.bya_COLOR[in_Offset_2] := Iby_Attr;

	in_Offset_1 := in_Offset_1 + INT#1;
	in_Offset_2 := in_Offset_2 + INT#1;

END_FOR;

(* linke obere Ecke ausgeben *)
in_Offset_1 := (Iin_Y1 * 80) + Iin_X1;
Xus_TN_SCREEN.bya_CHAR[in_Offset_1] := by_BorderChar_L_T;
Xus_TN_SCREEN.bya_COLOR[in_Offset_1] := Iby_Attr;

(* rechte obere Ecke ausgeben *)
in_Offset_1 := (Iin_Y1 * 80) + Iin_X2;
Xus_TN_SCREEN.bya_CHAR[in_Offset_1] := by_BorderChar_R_T;
Xus_TN_SCREEN.bya_COLOR[in_Offset_1] := Iby_Attr;

(* linke untere Ecke ausgeben *)
in_Offset_1 := (Iin_Y2 * 80) + Iin_X1;
Xus_TN_SCREEN.bya_CHAR[in_Offset_1] := by_BorderChar_R_B;
Xus_TN_SCREEN.bya_COLOR[in_Offset_1] := Iby_Attr;

(* rechte untere Ecke ausgeben *)
in_Offset_1 := (Iin_Y2 * 80) + Iin_X2;
Xus_TN_SCREEN.bya_CHAR[in_Offset_1] := by_BorderChar_L_B;
Xus_TN_SCREEN.bya_COLOR[in_Offset_1] := Iby_Attr;

(* revision history
ks	10. mai. 2010	rev 1.0
	original version
*)
END_FUNCTION_BLOCK

(* POU TN_SC_FILL, ST *)
FUNCTION_BLOCK TN_SC_FILL
VAR
	in_X : INT;
	in_Y : INT;
	in_Offset : INT;
END_VAR
VAR_INPUT
	Iin_Y1 : INT;
	Iin_X1 : INT;
	Iin_Y2 : INT;
	Iin_X2 : INT;
	Iby_CHAR : BYTE;
	Iby_Attr : BYTE;
END_VAR
VAR_IN_OUT
	Xus_TN_SCREEN : us_TN_SCREEN;
END_VAR

(*
version 1.0		10. mai 2010
programmer		ks
tested by		ks

TN_SC_FILL füllt einen rechteckigen Bereich mit einem Zeichen
*)
IF TN_SC_XY2_ERROR(Iin_X1,Iin_Y1,Iin_X2,Iin_Y2) THEN RETURN; END_IF;

FOR in_Y := Iin_Y1 TO Iin_Y2 DO
	Xus_TN_SCREEN.bya_Line_Update[in_Y] := TRUE; (* Zeile zum Updaten freigeben *)
	in_Offset := (in_Y * 80) + Iin_X1;
	FOR in_X := Iin_X1 TO Iin_X2 DO
		Xus_TN_SCREEN.bya_CHAR[in_Offset]  := Iby_CHAR; (* Zeichen eintragen *)
		Xus_TN_SCREEN.bya_COLOR[in_Offset] := Iby_Attr; (* Farbe eintragen *)
		in_Offset := in_Offset + 1;
	END_FOR;
END_FOR;

(* revision history
ks	10. mai. 2010	rev 1.0
	original version
*)
END_FUNCTION_BLOCK

(* POU TN_SC_WRITE_C, ST *)
FUNCTION_BLOCK TN_SC_WRITE_C
VAR
	FB_TN_SC_WRITE : TN_SC_WRITE;
END_VAR
VAR_INPUT
	Iin_Y : INT;
	Iin_X : INT;
	Iby_ATTR : BYTE;
	Ist_STRING : STRING;
	Iin_LENGTH : INT;
	Iin_OPTION : INT;
END_VAR
VAR_IN_OUT
	Xus_TN_SCREEN : us_TN_SCREEN;
END_VAR

(*
version 1.0		10. mai 2010
programmer		ks
tested by		ks

TN_SC_WRITE_C korrigiert die Textlänge und schreibt den Text an die angegebenen Koordinate
*)
(* Text ausgeben *)
FB_TN_SC_WRITE( Iin_Y := Iin_Y,
				Iin_X := Iin_X,
				Iby_ATTR := Iby_ATTR,
				Ist_STRING := FIX(str:=Ist_STRING,L:=Iin_LENGTH,C:=BYTE#32,M:=Iin_OPTION),
				Xus_TN_SCREEN := Xus_TN_SCREEN);

(* revision history
ks	10. mai. 2010	rev 1.0
	original version
*)
END_FUNCTION_BLOCK

(* POU TN_SC_WRITE, ST *)
FUNCTION_BLOCK TN_SC_WRITE
VAR
	bo_Color : BOOL;
	in_Offset : INT;
	in_Char_Index : INT;
	in_String_Length : INT;
END_VAR
VAR_INPUT
	Iin_Y : INT;
	Iin_X : INT;
	Iby_ATTR : BYTE;
	Ist_STRING : STRING;
END_VAR
VAR_IN_OUT
	Xus_TN_SCREEN : us_TN_SCREEN;
END_VAR

(*
version 1.0		10. mai 2010
programmer		ks
tested by		ks

TN_SC_WRITE schreibt einem Text an die angegebene Koordinate
*)
in_String_Length := LEN(Ist_STRING);
IF TN_SC_XY_ERROR(Iin_X + in_String_Length - 1,Iin_Y) THEN RETURN; END_IF;
Xus_TN_SCREEN.bya_Line_Update[Iin_Y] := TRUE; (* Zeile zum Updaten freigeben *)
in_Offset := (Iin_Y * 80) + Iin_X; (* Offset des ersten Zeichen berechnen *)
bo_Color := Iby_ATTR <> BYTE#00;

(* Zeichen und Attribute des String kopieren *)
FOR in_Char_Index := 1 TO in_String_Length DO
	IF bo_Color THEN Xus_TN_SCREEN.bya_COLOR[in_Offset] := Iby_ATTR; END_IF;
	Xus_TN_SCREEN.bya_CHAR[in_Offset] := CODE(STR:=Ist_STRING,POS:=in_Char_Index);
	in_Offset := in_Offset + INT#1;
END_FOR;

Xus_TN_SCREEN.in_EOS_Offset := in_Offset; (* End of String Offset sichern *)

(* revision history
ks	10. mai. 2010	rev 1.0
	original version
*)
END_FUNCTION_BLOCK

(* POU TN_SC_XY_ERROR, ST *)
FUNCTION TN_SC_XY_ERROR : BOOL
VAR_INPUT
	X : INT;
	Y : INT;
END_VAR

(*
version 1.0		10. mai 2010
programmer		ks
tested by		ks

TN_SC_XY_ERROR prüft ob die angegenene Koordinaten gültig sind 
*)
(* min und max werte prüfen *)
TN_SC_XY_ERROR := Y < 0 OR X < 0 OR Y > 23 OR X > 79;

(* revision history
ks	10. mai. 2010	rev 1.0
	original version
*)
END_FUNCTION

(* POU TN_INPUT_SELECT_TEXT, ST *)
FUNCTION_BLOCK TN_INPUT_SELECT_TEXT
VAR
	in_count : INT;
	by_Attr : BYTE;
	st_String : STRING;
END_VAR
VAR
	FB_TN_SC_WRITE : TN_SC_WRITE;
END_VAR
VAR_IN_OUT
	Xus_TN_SCREEN : us_TN_SCREEN;
	Xus_TN_INPUT_CONTROL_DATA : us_TN_INPUT_CONTROL_DATA;
END_VAR

(*
version 1.1		06. apr 2011
programmer		ks
tested by			ks

TN_SELECT_TEXT dient zur verwaltung und darstellung einer Elementeauswahl
*)
(* Benutzereingabe auswerten -> Selektion Text n *)
IF Xus_TN_INPUT_CONTROL_DATA.bo_Focus = TRUE THEN

(* Leertaste-Taste auswerten *)
	IF Xus_TN_INPUT_CONTROL_DATA.by_Input_ASCII_Code = BYTE#32 THEN
		Xus_TN_INPUT_CONTROL_DATA.in_selected := Xus_TN_INPUT_CONTROL_DATA.in_selected + INT#01; 
		Xus_TN_INPUT_CONTROL_DATA.bo_Update_Input := TRUE;
	END_IF;
 
	(* Return-Taste auswerten *)
	IF Xus_TN_INPUT_CONTROL_DATA.by_Input_Exten_Code = BYTE#13 THEN
		Xus_TN_INPUT_CONTROL_DATA.bo_Input_Entered := TRUE;
	END_IF;

END_IF;

(* Aktualisierung der Anzeige *)
IF (Xus_TN_INPUT_CONTROL_DATA.bo_Update_Input = TRUE) OR (Xus_TN_INPUT_CONTROL_DATA.bo_Update_All = TRUE) THEN

	(* Title-Text ausgeben *)
	IF Xus_TN_INPUT_CONTROL_DATA.bo_Update_All = TRUE THEN

		IF (Xus_TN_INPUT_CONTROL_DATA.in_Title_X_Offset = INT#00) AND (Xus_TN_INPUT_CONTROL_DATA.in_Title_Y_Offset = INT#00) THEN
			(* wenn Offset X,Y =0 dann Titlestring links vom Element positionieren *)
			FB_TN_SC_WRITE.Iin_Y := Xus_TN_INPUT_CONTROL_DATA.in_Y;
			FB_TN_SC_WRITE.Iin_X := Xus_TN_INPUT_CONTROL_DATA.in_X - LEN(Xus_TN_INPUT_CONTROL_DATA.st_Title_String);

		ELSE
			(* Title-Text durch Row, Color-Offset ausgeben *)
			FB_TN_SC_WRITE.Iin_Y := Xus_TN_INPUT_CONTROL_DATA.in_Y + Xus_TN_INPUT_CONTROL_DATA.in_Title_Y_Offset;
			FB_TN_SC_WRITE.Iin_X := Xus_TN_INPUT_CONTROL_DATA.in_X + Xus_TN_INPUT_CONTROL_DATA.in_Title_X_Offset;
		END_IF;

		(* Title-Text durch Row, Color-Offset ausgeben *)
		FB_TN_SC_WRITE(	Iby_ATTR := Xus_TN_INPUT_CONTROL_DATA.by_Title_Attr,
						Ist_STRING := Xus_TN_INPUT_CONTROL_DATA.st_Title_String,
						Xus_TN_SCREEN := Xus_TN_SCREEN);

	END_IF;

	(* Eingabezeile verarbeiten *)

	(* Anzahl der Elemente bestimmen *)
	in_count := ELEMENT_COUNT(SEP:=BYTE#35,ELEMENT:=Xus_TN_INPUT_CONTROL_DATA.st_Input_Data);

	IF in_Count > INT#00 THEN

		IF Xus_TN_INPUT_CONTROL_DATA.in_selected < INT#1 THEN
			Xus_TN_INPUT_CONTROL_DATA.in_selected := INT#01;
		END_IF;

		IF Xus_TN_INPUT_CONTROL_DATA.in_selected > in_count THEN
			Xus_TN_INPUT_CONTROL_DATA.in_selected := INT#01;
		END_IF;

		st_String := ELEMENT_GET(SEP:=BYTE#35,POS:=Xus_TN_INPUT_CONTROL_DATA.in_selected - 1,ELEMENT:=Xus_TN_INPUT_CONTROL_DATA.st_Input_Data);

		st_String := FIX(	str:=st_String,
							L:=LEN(Xus_TN_INPUT_CONTROL_DATA.st_Input_Mask),
							C:=BYTE#32,
							M:=Xus_TN_INPUT_CONTROL_DATA.in_Input_Option);

		Xus_TN_INPUT_CONTROL_DATA.st_Input_String := st_String;

		IF Xus_TN_INPUT_CONTROL_DATA.bo_Focus = TRUE THEN
			by_Attr := Xus_TN_INPUT_CONTROL_DATA.by_Attr_mF;
		ELSE
			by_Attr := Xus_TN_INPUT_CONTROL_DATA.by_Attr_oF;
		END_IF;

		FB_TN_SC_WRITE(	Iin_Y := Xus_TN_INPUT_CONTROL_DATA.in_Y,
						Iin_X := Xus_TN_INPUT_CONTROL_DATA.in_X,
						Iby_ATTR := by_Attr,
						Ist_STRING := st_String,
						Xus_TN_SCREEN := Xus_TN_SCREEN);
	END_IF;

	(* Cursor auf aktuelle Position setzen *)
	Xus_TN_INPUT_CONTROL_DATA.in_Cursor_Y := Xus_TN_INPUT_CONTROL_DATA.in_Y;
	Xus_TN_INPUT_CONTROL_DATA.in_Cursor_X := Xus_TN_INPUT_CONTROL_DATA.in_X;

	(* Update-Flag's rücksetzen *)
	Xus_TN_INPUT_CONTROL_DATA.bo_Update_All := FALSE;
	Xus_TN_INPUT_CONTROL_DATA.bo_Update_Input := FALSE;

END_IF;

(* revision history

ks	06. apr. 2011	rev 1.1
	list_len und list_get durch element_count und element_get ersetzt

ks	10. mai. 2010	rev 1.0
	original version
*)
END_FUNCTION_BLOCK

(* POU TN_INPUT_EDIT_LINE, ST *)
FUNCTION_BLOCK TN_INPUT_EDIT_LINE
VAR
	in_count : INT;
	in_Count_End : INT;
	in_CursorOffset : INT;
	by_Attr : BYTE;
	st_String : STRING;
	bo_Pos_Found : BOOL;
	st_CHAR : STRING(1);
	in_old_charpos : INT;
END_VAR
VAR
	FB_TN_SC_WRITE : TN_SC_WRITE;
END_VAR
VAR_IN_OUT
	Xus_TN_SCREEN : us_TN_SCREEN;
	Xus_TN_INPUT_CONTROL_DATA : us_TN_INPUT_CONTROL_DATA;
END_VAR

(*
version 1.0		10. mai 2010
programmer		ks
tested by		ks

TN_INPUT_EDIT_LINE ermöglicht die Eingabe von Texten durch eine Editierbare Eingabezeile
*)
(* Cursorsteuerung rücksetzen *)
in_CursorOffset := INT#0;

IF Xus_TN_INPUT_CONTROL_DATA.bo_Focus = TRUE THEN

	(* Texteingabe erkannt ? *)
	IF Xus_TN_INPUT_CONTROL_DATA.by_Input_ASCII_Code > BYTE#0 THEN

		IF (Xus_TN_INPUT_CONTROL_DATA.bo_Input_Only_Num = TRUE AND Xus_TN_INPUT_CONTROL_DATA.bo_Input_ASCII_IsNum = TRUE)
			OR (Xus_TN_INPUT_CONTROL_DATA.bo_Input_Only_Num = FALSE) THEN

			(* ASCII Wert in einen String wandeln *)
			st_CHAR := CHR_TO_STRING(C:=Xus_TN_INPUT_CONTROL_DATA.by_Input_ASCII_Code);

			(* Eingabe übernehmen *)
			Xus_TN_INPUT_CONTROL_DATA.st_Input_Data := REPLACE(Xus_TN_INPUT_CONTROL_DATA.st_Input_Data,
			st_CHAR,INT#1,Xus_TN_INPUT_CONTROL_DATA.in_Cursor_Pos);

			in_CursorOffset := INT#1;
			Xus_TN_INPUT_CONTROL_DATA.bo_Update_Input := TRUE;
		END_IF;
	END_IF;

	CASE BYTE_TO_INT(Xus_TN_INPUT_CONTROL_DATA.by_Input_Exten_Code) OF

	67: (* Cursor rechts gedrückt *)
		in_CursorOffset := INT#1;

	68: (* Cursor links gedrückt *)
		in_CursorOffset := -1;

	08: (* Backspace gedrückt *)
		Xus_TN_INPUT_CONTROL_DATA.st_Input_Data := REPLACE(Xus_TN_INPUT_CONTROL_DATA.st_Input_Data, ' ', 1,Xus_TN_INPUT_CONTROL_DATA.in_Cursor_Pos);
		Xus_TN_INPUT_CONTROL_DATA.bo_Update_Input := TRUE;
		in_CursorOffset := -1;

	13: (* Enter-Taste gedrückt *)
		IF LEN(Xus_TN_INPUT_CONTROL_DATA.st_Input_Mask) > INT#00 THEN
			(* Eingabestring übernehmen *)
			Xus_TN_INPUT_CONTROL_DATA.st_Input_String := Xus_TN_INPUT_CONTROL_DATA.st_Input_Data;

			(* Eingabestring -> links und rechts Leerzeichen entfernen *)
			Xus_TN_INPUT_CONTROL_DATA.st_Input_String := TRIME(str:=Xus_TN_INPUT_CONTROL_DATA.st_Input_String);
			Xus_TN_INPUT_CONTROL_DATA.bo_Input_Entered := TRUE;

			(* neue Eingabe vorbereiten *)
			Xus_TN_INPUT_CONTROL_DATA.st_Input_Data := Xus_TN_INPUT_CONTROL_DATA.st_Input_Mask;

			Xus_TN_INPUT_CONTROL_DATA.in_Cursor_Pos := INT#1;
			Xus_TN_INPUT_CONTROL_DATA.bo_Update_Input := TRUE;

			(* suche erstes Position in Eingabemaske *)
			st_CHAR := MID(Xus_TN_INPUT_CONTROL_DATA.st_Input_Mask,1,Xus_TN_INPUT_CONTROL_DATA.in_Cursor_Pos);
			IF st_CHAR <> ' ' THEN
				(* nächsten Eingabeposition suchen *)
				in_CursorOffset := INT#1;
			END_IF;
		END_IF;
	END_CASE;
END_IF;

(* Cursor richtung rechts bewegen                                   *)
IF (in_CursorOffset > INT#0) OR (Xus_TN_INPUT_CONTROL_DATA.in_Cursor_Pos = INT#0) THEN
	bo_Pos_Found := FALSE;

	in_Count := Xus_TN_INPUT_CONTROL_DATA.in_Cursor_Pos + INT#1;
	in_Count_End := LEN(Xus_TN_INPUT_CONTROL_DATA.st_Input_Mask);

	WHILE (in_count <= in_Count_End) AND (bo_Pos_Found = FALSE) DO

		st_CHAR := MID(Xus_TN_INPUT_CONTROL_DATA.st_Input_Mask,1,in_count);
		IF st_CHAR = ' ' THEN
			Xus_TN_INPUT_CONTROL_DATA.in_Cursor_Pos := in_count;
			Xus_TN_INPUT_CONTROL_DATA.bo_Update_Input := TRUE;
			bo_Pos_Found := TRUE;
		END_IF;

		in_count := in_count + INT#1;

	END_WHILE;
END_IF;

(* Cursor richtung links bewegen *)
IF in_CursorOffset < INT#0 THEN
	bo_Pos_Found := FALSE;

	in_Count     := Xus_TN_INPUT_CONTROL_DATA.in_Cursor_Pos - INT#01;
	in_Count_End := INT#1;

	WHILE (in_count >= in_Count_End) AND (bo_Pos_Found = FALSE) DO

		st_CHAR := MID(Xus_TN_INPUT_CONTROL_DATA.st_Input_Mask,1,in_count);
		IF st_CHAR = ' ' THEN
			Xus_TN_INPUT_CONTROL_DATA.in_Cursor_Pos := in_count;
			Xus_TN_INPUT_CONTROL_DATA.bo_Update_Input := TRUE;
			bo_Pos_Found := TRUE;
		END_IF;

		in_count := in_count - INT#1;
	END_WHILE;
END_IF;

(* maximale Cursorposition ? *)
IF Xus_TN_INPUT_CONTROL_DATA.in_Cursor_Pos > LEN(Xus_TN_INPUT_CONTROL_DATA.st_Input_Data) THEN
	Xus_TN_INPUT_CONTROL_DATA.in_Cursor_Pos := LEN(Xus_TN_INPUT_CONTROL_DATA.st_Input_Data);
	Xus_TN_INPUT_CONTROL_DATA.bo_Update_Input := TRUE;
END_IF;

(* minimale Cursorposition ? *)
IF Xus_TN_INPUT_CONTROL_DATA.in_Cursor_Pos < INT#1 THEN
	Xus_TN_INPUT_CONTROL_DATA.in_Cursor_Pos := INT#1;
	Xus_TN_INPUT_CONTROL_DATA.bo_Update_Input := TRUE;
END_IF;

(* Aktualisierung der Anzeige *)
IF (Xus_TN_INPUT_CONTROL_DATA.bo_Update_Input = TRUE) OR (Xus_TN_INPUT_CONTROL_DATA.bo_Update_All = TRUE) THEN

	(* Title-Text ausgeben *)
	IF (Xus_TN_INPUT_CONTROL_DATA.bo_Update_All = TRUE) THEN

		IF (Xus_TN_INPUT_CONTROL_DATA.in_Title_X_Offset = INT#00) AND (Xus_TN_INPUT_CONTROL_DATA.in_Title_Y_Offset = INT#00) THEN
			(* wenn Offset X,Y =0 dann Titlestring links vom Element positionieren *)
			FB_TN_SC_WRITE.Iin_Y := Xus_TN_INPUT_CONTROL_DATA.in_Y;
			FB_TN_SC_WRITE.Iin_X := Xus_TN_INPUT_CONTROL_DATA.in_X - LEN(Xus_TN_INPUT_CONTROL_DATA.st_Title_String);
		ELSE
			(* Title-Text durch Row, Color-Offset ausgeben *)
			FB_TN_SC_WRITE.Iin_Y := Xus_TN_INPUT_CONTROL_DATA.in_Y + Xus_TN_INPUT_CONTROL_DATA.in_Title_Y_Offset;
			FB_TN_SC_WRITE.Iin_X := Xus_TN_INPUT_CONTROL_DATA.in_X + Xus_TN_INPUT_CONTROL_DATA.in_Title_X_Offset;
		END_IF;

		(* Title-Text durch Row, Color-Offset ausgeben *)
		FB_TN_SC_WRITE(	Iby_ATTR := Xus_TN_INPUT_CONTROL_DATA.by_Title_Attr,
						Ist_STRING := Xus_TN_INPUT_CONTROL_DATA.st_Title_String,
						Xus_TN_SCREEN := Xus_TN_SCREEN);
	END_IF;

	(* Eingabetext ausgeben *)
	IF (Xus_TN_INPUT_CONTROL_DATA.bo_Input_Hidden = TRUE) THEN

		st_String := '';

		IF LEN(Xus_TN_INPUT_CONTROL_DATA.st_Input_Data) = LEN(Xus_TN_INPUT_CONTROL_DATA.st_Input_Mask) THEN
			(* Eingabemodus: HIDDEN *)
			FOR in_count := 1 TO LEN(Xus_TN_INPUT_CONTROL_DATA.st_Input_Data) DO

				(* Zeichen aus Eingabemaske lesen *)
				st_CHAR := MID(Xus_TN_INPUT_CONTROL_DATA.st_Input_Mask,1,in_count);

				(* Eingabe oder Maskenzeichen ausgeben *)
				IF st_CHAR = ' ' THEN

					(* Zeichen aus Eingabedata lesen *)
					st_CHAR := MID(Xus_TN_INPUT_CONTROL_DATA.st_Input_Data,1,in_count);

					IF st_CHAR = ' ' THEN
						(* Leerzeichen ausgeben *)
						st_String := CONCAT(st_String, ' ');

					ELSE
						(* verdecktes Zeichen ausgeben *)
						st_String := CONCAT(st_String, '*');

					END_IF;

				ELSE
					(* Zeichen aus Eingabemaske übernehmen *)
					st_CHAR := MID(Xus_TN_INPUT_CONTROL_DATA.st_Input_Data,1,in_count);
					st_String := CONCAT(st_String,st_CHAR);

				END_IF;
			END_FOR;
		END_IF;
	ELSE

		(* Eingabemodus: NORMAL *)
		st_String := Xus_TN_INPUT_CONTROL_DATA.st_Input_Data;

	END_IF;

	(* String ausgeben *)

	IF Xus_TN_INPUT_CONTROL_DATA.bo_Focus = TRUE THEN
		by_Attr := Xus_TN_INPUT_CONTROL_DATA.by_Attr_mF;
	ELSE
		by_Attr := Xus_TN_INPUT_CONTROL_DATA.by_Attr_oF;
	END_IF;

	FB_TN_SC_WRITE(	Iin_Y := Xus_TN_INPUT_CONTROL_DATA.in_Y,
					Iin_X := Xus_TN_INPUT_CONTROL_DATA.in_X,
					Iby_ATTR := by_Attr,
					Ist_STRING := st_String,
					Xus_TN_SCREEN := Xus_TN_SCREEN);

	(* Cursor auf aktuelle Position setzen *)
	Xus_TN_INPUT_CONTROL_DATA.in_Cursor_Y := Xus_TN_INPUT_CONTROL_DATA.in_Y;
	Xus_TN_INPUT_CONTROL_DATA.in_Cursor_X := Xus_TN_INPUT_CONTROL_DATA.in_X + Xus_TN_INPUT_CONTROL_DATA.in_Cursor_Pos - INT#1;

	in_old_charpos := INT#0;

	(* Update-Flag's rücksetzen *)
	Xus_TN_INPUT_CONTROL_DATA.bo_Update_All := FALSE;
	Xus_TN_INPUT_CONTROL_DATA.bo_Update_Input := FALSE;
END_IF;

(* revision history
ks	10. mai. 2010	rev 1.0
	original version
*)
END_FUNCTION_BLOCK

(* POU TN_INPUT_MENU_BAR, ST *)
FUNCTION_BLOCK TN_INPUT_MENU_BAR
VAR
	FB_TN_INPUT_MENU_POPUP : TN_INPUT_MENU_POPUP;
	us_TN_MENU_POPUP : us_TN_MENU_POPUP;
	FB_TN_SC_WRITE_C : TN_SC_WRITE_C;
END_VAR
VAR
	in_ROW : INT;
	in_COL : INT;
	in_TITLE_Length : INT;
	st_MENU_BAR : STRING(STRING_LENGTH);
	st_MENU_TITLE : STRING;
	in_Count : INT;
	in_Index : INT;
	by_New_KeyCode : BYTE;
	in_Scroll_Offset : INT;
	by_ATTR : BYTE;
	bo_Reset_Position :	BOOL;
END_VAR
VAR_IN_OUT
	Xus_TN_MENU : us_TN_MENU;
	Xus_TN_SCREEN : us_TN_SCREEN;
END_VAR

(*
version 1.1		06. apr 2011
programmer		ks
tested by			ks

TN_MENU_BAR ermöglicht die verwaltung und darstellung einer MENU-BAR
*)
(* sicherstellen das rechteck immer innerhalb screen positioniert wird *)

IF (Xus_TN_MENU.in_State = INT#00) AND (Xus_TN_MENU.bo_Create = TRUE) THEN
	Xus_TN_MENU.in_State := INT#01;
	Xus_TN_MENU.bo_Create := FALSE;
	Xus_TN_MENU.in_Menu_Selected := INT#00;
	Xus_TN_MENU.bo_Update := TRUE;
	bo_Reset_Position := TRUE;

	(* Menu-Bar - Hauptmenue *)
	st_MENU_BAR := ELEMENT_GET(SEP:=BYTE#37,POS:=0,ELEMENT:=Xus_TN_MENU.st_MENU_TEXT);

	(* Menu-Bar - Anzahl der Elemente bestimmen *)
	Xus_TN_MENU.in_Menu_E_Count := ELEMENT_COUNT(SEP:=BYTE#35,ELEMENT:=st_MENU_BAR);

END_IF;

(* Keycode ablegen *)
by_New_KeyCode := Xus_TN_SCREEN.by_Input_Exten_Code;

(* Popup-Menu Tastensteuerung (nur Cursor oben + unten zulassen *)
IF (by_New_KeyCode = BYTE#65) OR (by_New_KeyCode = BYTE#66) THEN
	us_TN_MENU_POPUP.by_Input_Exten_Code := by_New_KeyCode;
ELSE
	us_TN_MENU_POPUP.by_Input_Exten_Code := BYTE#00;
END_IF;

(* Escape *)
IF (by_New_KeyCode = BYTE#27) THEN
	(* Menu war inaktiv -> Escape -> Menu aktivieren *)
	IF (Xus_TN_MENU.in_State = INT#01) AND (Xus_TN_SCREEN.bo_Modal_Dialog = FALSE) THEN
		Xus_TN_MENU.in_State := INT#02;
		Xus_TN_MENU.bo_Update := TRUE;
		Xus_TN_MENU.in_Menu_Selected := INT#00;

		Xus_TN_SCREEN.bo_Menue_Bar_Dialog := TRUE;

		(* Menu war aktiv -> Escape -> Menu deaktivieren *)
	ELSIF (Xus_TN_MENU.in_State = INT#02) THEN
		us_TN_MENU_POPUP.bo_Destroy := TRUE;
		Xus_TN_MENU.bo_Update := TRUE;
		Xus_TN_MENU.in_State := INT#01;
		bo_Reset_Position := TRUE;

		Xus_TN_SCREEN.bo_Menue_Bar_Dialog := FALSE;
	END_IF;
END_IF;

(* Menu aktiv *)
IF (Xus_TN_MENU.in_State = INT#02) THEN

	(* Return *)
	IF (by_New_KeyCode = BYTE#13)  THEN
		us_TN_MENU_POPUP.bo_Destroy := TRUE;
		Xus_TN_MENU.bo_Update := TRUE;
		Xus_TN_MENU.in_State := INT#01;
		bo_Reset_Position := TRUE;
		Xus_TN_MENU.in_Menu_Selected := (Xus_TN_MENU.in_Cur_Menu_Item * INT#10) + Xus_TN_MENU.in_Cur_Sub_Item;
		Xus_TN_SCREEN.by_Input_Exten_Code := BYTE#00;

		Xus_TN_SCREEN.bo_Menue_Bar_Dialog := FALSE;

		(* Destroy-Befehl -> Popup-Menu beenden *)
	ELSIF (Xus_TN_MENU.bo_Destroy = TRUE) THEN
		us_TN_MENU_POPUP.bo_Destroy := TRUE;
		Xus_TN_MENU.bo_Update := TRUE;
		Xus_TN_MENU.in_State := INT#01;
		bo_Reset_Position := TRUE;
		Xus_TN_MENU.in_Menu_Selected := INT#00;
		Xus_TN_SCREEN.by_Input_Exten_Code := BYTE#00;

		Xus_TN_SCREEN.bo_Menue_Bar_Dialog := FALSE;

	END_IF;

	IF (by_New_KeyCode = BYTE#67) THEN (* Cursor rechts *)
		in_Scroll_Offset := INT#1;
		Xus_TN_MENU.bo_Update := TRUE;
		Xus_TN_SCREEN.by_Input_Exten_Code := BYTE#00;

	ELSIF (by_New_KeyCode = BYTE#68) THEN (* Cursor links *)
		in_Scroll_Offset := -1;
		Xus_TN_MENU.bo_Update := TRUE;
		Xus_TN_SCREEN.by_Input_Exten_Code := BYTE#00;
	END_IF;
END_IF;

IF bo_Reset_Position = TRUE THEN
	bo_Reset_Position := FALSE;
	Xus_TN_MENU.in_X_SM_old := -1;
	Xus_TN_MENU.in_Y_SM_old := -1;
	Xus_TN_MENU.in_X_SM_new := -1;
	Xus_TN_MENU.in_Y_SM_new := -1;
END_IF;

(* POPUP-Menu updaten *)
IF (Xus_TN_MENU.in_State > INT#00) AND (Xus_TN_MENU.bo_Update = TRUE) THEN

	Xus_TN_MENU.bo_Update := FALSE; 

	in_ROW := Xus_TN_MENU.in_Y;
	in_COL := Xus_TN_MENU.in_X;

	(* Scrolloffset *)
	IF in_Scroll_Offset <> INT#00 THEN
		Xus_TN_MENU.in_Cur_Menu_Item := INC2(Xus_TN_MENU.in_Cur_Menu_Item,in_Scroll_Offset,1,Xus_TN_MENU.in_Menu_E_Count);
		in_Scroll_Offset := INT#00;
	ELSE
		(* Item = 0 und kein Scrolloffset *)
		IF (Xus_TN_MENU.in_Cur_Menu_Item = INT#00) THEN
			Xus_TN_MENU.in_Cur_Menu_Item := INT#01;
		END_IF;
	END_IF;

	(* alle Menutext zeichnen *)
	FOR in_Count := INT#01 TO Xus_TN_MENU.in_Menu_E_Count DO;

		(* Zeichenfarbe bestimmen *)
		IF (in_Count = Xus_TN_MENU.in_Cur_Menu_Item) AND (Xus_TN_MENU.in_State > INT#01 ) THEN
			by_ATTR := Xus_TN_MENU.by_Attr_mF;

			Xus_TN_MENU.in_Y_SM_new := in_ROW + INT#01;
			Xus_TN_MENU.in_X_SM_new := in_COL;

		ELSE
			by_ATTR := Xus_TN_MENU.by_Attr_oF;
		END_IF;

		st_MENU_TITLE := ELEMENT_GET(SEP:=BYTE#35,POS:=in_Count - 1,ELEMENT:=st_MENU_BAR);

		in_TITLE_Length := LEN(st_MENU_TITLE) + INT#02;

		FB_TN_SC_WRITE_C(	Iin_Y := in_ROW,
							Iin_X := in_COL,
							Iby_ATTR := by_ATTR,
							Iin_LENGTH := in_TITLE_Length,
							Iin_OPTION := INT#02,
							Ist_STRING := st_MENU_TITLE,
							Xus_TN_SCREEN := Xus_TN_SCREEN);

		in_COL := in_COL + in_TITLE_Length;

	END_FOR;
END_IF;

IF Xus_TN_MENU.in_X_SM_new <> Xus_TN_MENU.in_X_SM_old THEN

	(* SubMenu ist aktiv -> beenden                                     *)
	IF us_TN_MENU_POPUP.bo_Activ = TRUE THEN
		us_TN_MENU_POPUP.bo_Destroy := TRUE;

		(* Sub-Menu bearbeiten *)
		FB_TN_INPUT_MENU_POPUP(	Xus_TN_MENU_POPUP := us_TN_MENU_POPUP,
								Xus_TN_SCREEN := Xus_TN_SCREEN);
	END_IF;

	IF us_TN_MENU_POPUP.bo_Activ = FALSE THEN
		(* Popup-Menu zu aktuellen Menu parametrieren und ausführen         *)
		in_Index := Xus_TN_MENU.in_Cur_Menu_Item;

		us_TN_MENU_POPUP.in_Y := Xus_TN_MENU.in_Y_SM_new;
		us_TN_MENU_POPUP.in_X := Xus_TN_MENU.in_X_SM_new;
		us_TN_MENU_POPUP.by_Attr_mF := Xus_TN_MENU.by_Attr_mF;
		us_TN_MENU_POPUP.by_Attr_oF := Xus_TN_MENU.by_Attr_oF;
		us_TN_MENU_POPUP.st_Menu_Text := ELEMENT_GET(SEP:=BYTE#37,POS:=in_Index,ELEMENT:=Xus_TN_MENU.st_MENU_TEXT);
		us_TN_MENU_POPUP.bo_Create := TRUE;

		Xus_TN_MENU.in_X_SM_old := Xus_TN_MENU.in_X_SM_new;
		Xus_TN_MENU.in_Y_SM_old := Xus_TN_MENU.in_Y_SM_new;

	END_IF;
END_IF;

(* Popup-Menu zyklisch aufrufen *)
FB_TN_INPUT_MENU_POPUP(	Xus_TN_MENU_POPUP := us_TN_MENU_POPUP,
						Xus_TN_SCREEN := Xus_TN_SCREEN);

(* aktuelles Item vom Popup-Menu kopieren *)
Xus_TN_MENU.in_Cur_Sub_Item := us_TN_MENU_POPUP.in_Cur_Item;

(* Destroy-Befehl *)
IF (Xus_TN_MENU.in_State = INT#01) THEN
	IF (Xus_TN_MENU.bo_Destroy = TRUE) THEN
		Xus_TN_MENU.in_State := INT#00;
		Xus_TN_MENU.bo_Destroy := FALSE;
		Xus_TN_MENU.in_Cur_Menu_Item := INT#00;
		Xus_TN_MENU.in_Cur_Sub_Item := INT#00;
	END_IF;
END_IF;

(* revision history
ks	06. apr. 2011	rev 1.1
	list_len und list_get durch element_count und element_get ersetzt

ks	10. mai. 2010	rev 1.0
	original version
*)
END_FUNCTION_BLOCK

(* POU TN_RECEIVE, ST *)
FUNCTION_BLOCK TN_RECEIVE
VAR_IN_OUT
	R_BUF :	NETWORK_BUFFER;
	Xus_TN_SCREEN : us_TN_SCREEN;
END_VAR
VAR
	REQ_Size : UINT;
	REQ1 : BYTE;
	REQ2 : BYTE;
	REQ3 : BYTE;
END_VAR

(*
version 1.0		10. mai 2010
programmer		ks
tested by		ks

TN_RECEIVE empfängt Tastatureingaben vom Telnet Client und wertet diese aus
*)
(* Datenempfang auswertung *)
Xus_TN_SCREEN.by_Input_ASCII_Code := BYTE#00;
Xus_TN_SCREEN.by_Input_Exten_Code := BYTE#00;

IF R_BUF.SIZE > UINT#0 THEN
	(* empfangene Daten auswerten *)
	REQ_Size := R_BUF.SIZE;
	REQ1 := R_BUF.BUFFER[0];
	REQ2 := R_BUF.BUFFER[1];
	REQ3 := R_BUF.BUFFER[2];

	IF REQ1 = BYTE#27 AND REQ_Size >= UINT#3 THEN (* Escape *)
		IF REQ2 = BYTE#91 THEN (* Cursor code *)
			IF (REQ3 >= BYTE#65 AND REQ3 <= BYTE#68) OR (REQ3 = BYTE#72) OR (REQ3 = BYTE#75) THEN (* 65..68 = Cursor o,u,r,l / 72 = POS1 / 75 = ENDE *)
				Xus_TN_SCREEN.by_Input_Exten_Code := REQ3;
			END_IF;
		ELSIF REQ2 = BYTE#79 THEN (* Sondertasten F1/F2/F3/F4 *)
			IF REQ3 >= BYTE#80 AND REQ3 <= BYTE#83 THEN
				Xus_TN_SCREEN.by_Input_Exten_Code := REQ3;
			END_IF;
		END_IF;
	ELSIF REQ1 >= BYTE#32 AND REQ1 <= BYTE#126 THEN
		Xus_TN_SCREEN.by_Input_ASCII_Code := REQ1;
		Xus_TN_SCREEN.bo_Input_ASCII_IsNum := ISC_NUM(REQ1); (* Auswertung auf Zahleneingabe *)
	ELSIF REQ1 = BYTE#8 OR REQ1 = BYTE#9 OR REQ1 = BYTE#13 OR REQ1 = BYTE#27 THEN (* prüfe auf Steuerzeichen 8=Backspace / 9=Tabulator / 13=Return / 27=Escape *)
		Xus_TN_SCREEN.by_Input_Exten_Code := REQ1;
	END_IF;

	(* Empfangsbuffer Datenlänge null eintragen (Telegramm zerstören *)
	R_BUF.SIZE := UINT#00;
END_IF;

(* revision history
ks	10. mai. 2010	rev 1.0
	original version
*)
END_FUNCTION_BLOCK

(* POU TN_SEND_ROWS, ST *)
FUNCTION_BLOCK TN_SEND_ROWS
VAR_IN_OUT
	IP_C : IP_C;
	S_BUF : NETWORK_BUFFER;
	Xus_TN_SCREEN : us_TN_SCREEN;
END_VAR
VAR_INPUT
	S_BUF_SIZE : INT;
END_VAR
VAR
	in_Line_Count : INT;(*Zähler um max alle 24 Zeilen zu durchlaufen*)
	in_Col_Count : INT;
	in_Last_Row_Index : INT;
	bo_Break_Loop : BOOL;
	in_Row_Count : INT;
	in_Offset : INT;
	in_Write_Index : INT;
	in_Write_Index_Backup : INT;
	by_Cur_Color : BYTE;
	by_last_Color : BYTE;
	in_Write_Stop : INT;
END_VAR

(*
version 1.0		10. mai 2010
programmer		ks
tested by		ks

TN_SEND_ROWS prüft den Bildschirmspeicher auf änderungen, und sendet diese zeilenweise an den Telnet Client 
*)
(* Verbindung vorhanden und kein Datensenden aktiv *)
IF (IP_C.C_STATE < BYTE#127 OR S_BUF.SIZE > UINT#0) THEN
	RETURN; (* nein -> Baustein beenden *)
END_IF;

(* aktuellen Schreibindex laden *)
in_Write_Index := UINT_TO_INT(S_BUF.SIZE) - 1;

(* aktuellen Schreibindex zwischenspeichern *)
in_Write_Index_Backup := in_Write_Index;

(* positive Flanke Connect on *)
IF (IP_C.C_STATE = BYTE#254) OR (Xus_TN_SCREEN.bo_Clear_Screen) THEN

	(* Clear-Screen Meldung rücksetzen *)
	Xus_TN_SCREEN.bo_Clear_Screen := FALSE;

	(* alle Zeilen für Update markieren *)
	FOR in_Line_Count := INT#00 TO INT#23 DO
		Xus_TN_SCREEN.bya_Line_Update[in_Line_Count] := TRUE;
	END_FOR;

	(* ESC [0;30,40m  Reset Attributes + Black,Black *)
	in_Write_Index := in_Write_Index + INT#1;
	S_BUF.BUFFER[in_Write_Index] := BYTE#16#1B; (* ESC *)
	in_Write_Index := in_Write_Index + INT#1;
	S_BUF.BUFFER[in_Write_Index] := BYTE#16#5B; (* [ *)
	in_Write_Index := in_Write_Index + INT#1;
	S_BUF.BUFFER[in_Write_Index] := BYTE#16#30; (* 0 *)
	in_Write_Index := in_Write_Index + INT#1;
	S_BUF.BUFFER[in_Write_Index] := BYTE#16#3B; (* ; *)
	in_Write_Index := in_Write_Index + INT#1;
	S_BUF.BUFFER[in_Write_Index] := BYTE#16#33; (* 3 *)

	(* Einerstelle Farbe Foreground ausgeben *)
	in_Write_Index := in_Write_Index + INT#1;
	S_BUF.BUFFER[in_Write_Index] := (SHR(Xus_TN_SCREEN.by_Clear_Screen_Attr,4) OR BYTE#16#30);

	in_Write_Index := in_Write_Index + INT#1;
	S_BUF.BUFFER[in_Write_Index] := BYTE#16#3B; (* ; *)
	in_Write_Index := in_Write_Index + INT#1;
	S_BUF.BUFFER[in_Write_Index] := BYTE#16#34; (* 4 *)

	(* Einerstelle Farbe Background ausgeben *)
	in_Write_Index := in_Write_Index + INT#1;
	S_BUF.BUFFER[in_Write_Index] := ((Xus_TN_SCREEN.by_Clear_Screen_Attr AND BYTE#16#07) OR BYTE#16#30);

	in_Write_Index := in_Write_Index + INT#1;
	S_BUF.BUFFER[in_Write_Index] := BYTE#16#6D; (* m *)

	(* ESC[2J Clear screen and home cursor *)
	in_Write_Index := in_Write_Index + INT#1;
	S_BUF.BUFFER[in_Write_Index] := BYTE#16#1B; (* ESC *)
	in_Write_Index := in_Write_Index + INT#1;
	S_BUF.BUFFER[in_Write_Index] := BYTE#16#5B; (* [ *)
	in_Write_Index := in_Write_Index + INT#1;
	S_BUF.BUFFER[in_Write_Index] := BYTE#16#32; (* 2 *)
	in_Write_Index := in_Write_Index + INT#1;
	S_BUF.BUFFER[in_Write_Index] := BYTE#16#4A; (* J *)

	(* ESC [?7l Off *)
	in_Write_Index := in_Write_Index + INT#1;
	S_BUF.BUFFER[in_Write_Index] := BYTE#16#1B; (* ESC *)
	in_Write_Index := in_Write_Index + INT#1;
	S_BUF.BUFFER[in_Write_Index] := BYTE#16#5B; (* [ *)
	in_Write_Index := in_Write_Index + INT#1;
	S_BUF.BUFFER[in_Write_Index] := BYTE#16#3F; (* ? *)
	in_Write_Index := in_Write_Index + INT#1;
	S_BUF.BUFFER[in_Write_Index] := BYTE#16#37; (* 7 *)
	in_Write_Index := in_Write_Index + INT#1;
	S_BUF.BUFFER[in_Write_Index] := BYTE#16#6C; (* l *)

END_IF;

in_Last_Row_Index := INT#0;
bo_Break_Loop := FALSE;
in_Write_Stop := S_BUF_SIZE - 20;

(* alle Zeilen durchlaufen *)
FOR in_Line_Count := 0 TO 23 DO

	in_Offset := in_Row_Count * INT#80;

	(* prüfen ob Update einer Zeile notwendig ist bzw. nach Reconnect *)
	IF (Xus_TN_SCREEN.bya_Line_Update[in_Row_Count] = TRUE) THEN

		(* Schreib-Cursor positionieren *)
		in_Write_Index := in_Write_Index + INT#1;
		S_BUF.BUFFER[in_Write_Index] := BYTE#16#1B; (* ESC *)
		in_Write_Index := in_Write_Index + INT#1;
		S_BUF.BUFFER[in_Write_Index] := BYTE#16#5B; (* [ *)

		(* Zehnerstelle Zeilennummer ausgeben *)
		in_Write_Index := in_Write_Index + INT#1;
		S_BUF.BUFFER[in_Write_Index] :=
		SHR(INT_TO_BCDC(in_Row_Count + INT#1),INT#4) OR BYTE#16#30;

		(* Einerstelle Zeilennummer ausgeben *)
		in_Write_Index := in_Write_Index + INT#1;
		S_BUF.BUFFER[in_Write_Index] :=
		(INT_TO_BCDC(in_Row_Count + INT#1) AND BYTE#16#0F) OR BYTE#16#30;

		in_Write_Index := in_Write_Index + INT#1;
		S_BUF.BUFFER[in_Write_Index] := BYTE#16#3B; (* ; *)
		in_Write_Index := in_Write_Index + INT#1;
		S_BUF.BUFFER[in_Write_Index] := BYTE#16#31; (* 1 *)
		in_Write_Index := in_Write_Index + INT#1;
		S_BUF.BUFFER[in_Write_Index] := BYTE#16#48; (* H *)

		(* alle Spalten einer Zeile durchlaufen *)
		FOR in_Col_Count := 0 TO 79 DO

			(* aktuelle Farbe bestimmen *)
			by_Cur_Color := Xus_TN_SCREEN.bya_COLOR[in_Offset];
			IF (by_Cur_Color <> by_last_Color) OR (in_Col_Count = INT#00) THEN

				(* Farbeinstellung: ANSI-Sequenz ESC[X;Y;Zm ausgeben *)
				in_Write_Index := in_Write_Index + INT#1;
				S_BUF.BUFFER[in_Write_Index] := BYTE#16#1B; (* ESC *)

				in_Write_Index := in_Write_Index + INT#1;
				S_BUF.BUFFER[in_Write_Index] := BYTE#16#5B; (* [ *)

				(* Farbeinstellung: dunkel oder Hell und blinken bestimmen *)

					IF (((by_Cur_Color AND BYTE#2#10001000) XOR (by_last_Color AND BYTE#2#10001000)) <> BYTE#00) OR (in_Col_Count = 0) THEN

						in_Write_Index := in_Write_Index + INT#1;
						S_BUF.BUFFER[in_Write_Index] := BYTE#16#30; (* 0 *)
						in_Write_Index := in_Write_Index + INT#1;
						S_BUF.BUFFER[in_Write_Index] := BYTE#16#3B; (* ; *)

						(* keine dunklen Farben gewünscht -> dann Bold & Bright *)
						IF (by_Cur_Color AND BYTE#2#00001000) = BYTE#2#00000000 THEN

							(* auf Bold & Btight Farben umstellen *)
							in_Write_Index := in_Write_Index + INT#1;
							S_BUF.BUFFER[in_Write_Index] := BYTE#16#31; (* 1 *) 
							in_Write_Index := in_Write_Index + INT#1;
							S_BUF.BUFFER[in_Write_Index] := BYTE#16#3B; (* ; *)

						END_IF;

						(* blinkenden Farben gewünscht *)
						IF (by_Cur_Color AND BYTE#2#10000000) = BYTE#2#10000000 THEN 

							(* auf Bold & Bright Farben umstellen *)
							in_Write_Index := in_Write_Index + INT#1;
							S_BUF.BUFFER[in_Write_Index] := BYTE#16#35; (* 5 *) 
							in_Write_Index := in_Write_Index + INT#1;
							S_BUF.BUFFER[in_Write_Index] := BYTE#16#3B; (* ; *)

						END_IF;

					END_IF;

					(* Zehnerstelle Farbe Foreground ausgeben *)
					in_Write_Index := in_Write_Index + INT#1;
					S_BUF.BUFFER[in_Write_Index] := BYTE#16#33; (* 3 *)

					(* Einerstelle Farbe Foreground ausgeben *)
					in_Write_Index := in_Write_Index + INT#1;
					S_BUF.BUFFER[in_Write_Index] := ((SHR(by_Cur_Color,4) AND BYTE#2#00000111) OR BYTE#16#30);

					in_Write_Index := in_Write_Index + INT#1;
					S_BUF.BUFFER[in_Write_Index] := BYTE#16#3B; (* ; *)

					(* Zehnerstelle Farbe Background ausgeben *)
					in_Write_Index := in_Write_Index + INT#1;
					S_BUF.BUFFER[in_Write_Index] := BYTE#16#34; (* 4 *)

					(* Einerstelle Farbe Background ausgeben *)
					in_Write_Index := in_Write_Index + INT#1;
					S_BUF.BUFFER[in_Write_Index] := ((by_Cur_Color AND BYTE#2#00000111) OR BYTE#16#30); 

					in_Write_Index := in_Write_Index + INT#1;
					S_BUF.BUFFER[in_Write_Index] := BYTE#16#6D; (* m *)

					(* neue Farbe als letzt verwendete speichern *)
					by_last_Color := by_Cur_Color;

				END_IF;

				(* Buffer Ende vorzeitig erreicht -> Ende *)
				IF (in_Write_Index > in_Write_Stop) THEN

					bo_Break_Loop := TRUE;
					EXIT;

				END_IF;

				(* ein TEXT-Zeichen von Screenbuffer in den Sendebuffer übertragen *)
				in_Write_Index := in_Write_Index + INT#1;
				S_BUF.BUFFER[in_Write_Index] := Xus_TN_SCREEN.bya_CHAR[in_Offset];

				(* nächste Spalte anwählen *)
				in_Offset := in_Offset + INT#01;
			END_FOR;

			IF (bo_Break_Loop = TRUE) THEN;

				(* Buffer Ende vorzeitig erreicht -> nur bis zur letzten kompletten Zeile uebertragen *)
				in_Write_Index := in_Last_Row_Index;

				EXIT;
			END_IF;

			(* Buffer ist noch nicht voll -> neue Zeile ubernehmen *)
			in_Last_Row_Index := in_Write_Index;
			Xus_TN_SCREEN.bya_Line_Update[in_Row_Count] := FALSE;

		END_IF;

		(* naechste Zeile adressieren *)
		in_Row_Count := in_Row_Count + INT#01;

		(* ab letzter Zeile wieder von vorne beginnen *)
		IF (in_Row_Count > INT#23) THEN
			in_Row_Count := INT#00;
		END_IF;
		(*-----------------------------------------------*)


	END_FOR;

	(* wenn in einen Update-Zyklus alle Zeilen auf einmal geschafft wurden *)
	(* wird der Row_Count auf ersten Zeile gestellt *)
	(* soll das hässliche Grafikflackern verhindern *)
	(* ansonsten wird bei der letzen Zeile weitergemacht *)
	IF (bo_Break_Loop = FALSE) THEN
		in_Row_Count := INT#00;
	END_IF;

	(* Edit-Cursor positionieren *)
	IF (in_Write_Index <> in_Write_Index_Backup) THEN

		in_Write_Index := in_Write_Index + INT#1;
		S_BUF.BUFFER[in_Write_Index] := BYTE#16#1B; (* ESC *)
		in_Write_Index := in_Write_Index + INT#1;
		S_BUF.BUFFER[in_Write_Index] := BYTE#16#5B; (* [ *)

		(* Zehnerstelle Zeilennummer ausgeben *)
		in_Write_Index := in_Write_Index + INT#1;
		S_BUF.BUFFER[in_Write_Index] := SHR(INT_TO_BCDC(Xus_TN_SCREEN.in_Cursor_Y + 1),INT#4) OR BYTE#16#30;

		(* Einerstelle Zeilennummer ausgeben *)
		in_Write_Index := in_Write_Index + INT#1;
		S_BUF.BUFFER[in_Write_Index] := (INT_TO_BCDC(Xus_TN_SCREEN.in_Cursor_Y + 1) AND BYTE#16#0F) OR BYTE#16#30;

		in_Write_Index := in_Write_Index + INT#1;
		S_BUF.BUFFER[in_Write_Index] := BYTE#16#3B; (* ; *)

		(* Zehnerstelle Spaltenummer ausgeben *)
		in_Write_Index := in_Write_Index + INT#1;
		S_BUF.BUFFER[in_Write_Index] := SHR(INT_TO_BCDC(Xus_TN_SCREEN.in_Cursor_X + 1),INT#4) OR BYTE#16#30;

		(* Einerstelle Spaltennummer ausgeben *)
		in_Write_Index := in_Write_Index + INT#1;
		S_BUF.BUFFER[in_Write_Index] := (INT_TO_BCDC(Xus_TN_SCREEN.in_Cursor_X + 1) AND BYTE#16#0F) OR BYTE#16#30;

		in_Write_Index := in_Write_Index + INT#1;
		S_BUF.BUFFER[in_Write_Index] := BYTE#16#48; (* H *)

END_IF;

(* aktuellen Schreibindex speichern -> Senden anstossen *)
S_BUF.SIZE := INT_TO_UINT(in_Write_Index + 1);

(* revision history
ks	10. mai. 2010	rev 1.0
	original version
*)
END_FUNCTION_BLOCK

(* POU LOG_VIEWPORT, ST *)
FUNCTION_BLOCK LOG_VIEWPORT
VAR_IN_OUT
	LC : LOG_CONTROL;
	LV : us_LOG_VIEWPORT;
END_VAR
VAR
	pos : INT;
	count : INT;
	idx : INT;
	base : INT;
	update_pos : BOOL;
END_VAR

(*
version 1.1		05 mai 2012
programmer		ks
tested BY		ks

LOG_VIEWPORT erzeugt einen Liste der Meldungen des Loggingbuffers die innerhalb einer virtuellen Ansicht enthalten sind.
*)
(* Scroll Button verarbeiten *)
IF LV.MOVE_TO_X <> 0 THEN
	CASE LV.MOVE_TO_X OF
	30000: pos := 1 ; (* älteste Meldung anzeigen *)
	30001: pos := LC.SIZE; (* neueste Meldung anzeigen *)
	30002: pos := pos + LV.COUNT; (* eine Seite nach unten blättern -> Richtung neuere Nachrichten *)
	30003: pos := pos - LV.COUNT; (* eine Seite nach oben blättern -> Richtung ältere Nachrichten *)
	ELSE
		pos := pos + LV.MOVE_TO_X;
	END_CASE;
	update_pos := TRUE;
	LV.MOVE_TO_X := 0;
END_IF;

IF (LV.UPDATE_COUNT <> LC.UPDATE_COUNT) OR update_pos THEN (* Aktualisierung überwachen *)
	LV.UPDATE := TRUE;
	LV.UPDATE_COUNT := LC.UPDATE_COUNT;
	update_pos := FALSE;

	(* pos prüfen und übernehmen *)
	IF LC.RING_MODE THEN
		pos := LIMIT(1,pos,LC.SIZE - LV.COUNT + 1);
	ELSE
		IF LC.IDX > LV.COUNT THEN
			pos := LIMIT(1,pos,LC.IDX - LV.COUNT + 1);
		ELSE
			pos := 1;
		END_IF;
	END_IF;

	(* idxBasis berechnen *)
	base := LC.IDX - pos - LV.COUNT + 1;
	IF LC.RING_MODE THEN 
		(* Anzeige im Ringpuffermodus *)
		FOR count:= 1 TO LV.COUNT DO
			idx := base + count;
			IF idx < 1 THEN
				idx := idx + LC.SIZE;
			END_IF;
			LV.LINE_ARRAY[count] := idx;
		END_FOR;
	ELSE
		(* Anzeige im Normalmodus *)
		FOR count:= 1 TO LV.COUNT DO
			idx := base + count;
			IF idx < 1 THEN
				(* Leere Zeile ausgeben *)
				LV.LINE_ARRAY[count] := 0;
			ELSE
				LV.LINE_ARRAY[count] := idx;
			END_IF;
		END_FOR;
	END_IF;
END_IF;

(* revision history
ks	01. mai 2010	rev 1.0
	original version

ks	05. mai 2012	rev 1.1
	Fehler im Ringmodus

*)
END_FUNCTION_BLOCK

(* POU TN_SC_VIEWPORT, ST *)
FUNCTION_BLOCK TN_SC_VIEWPORT
VAR
	FB_TN_SC_WRITE : TN_SC_WRITE;
	FB_TON : TON;
END_VAR
VAR
	in_index : INT;
	in_Color : INT;
	by_Attr : BYTE;
	in_count : INT;
END_VAR
VAR_IN_OUT
	Xus_LOG_VIEWPORT : us_LOG_VIEWPORT;
	Xus_LOG_CONTROL : LOG_CONTROL;
	Xus_TN_SCREEN : us_TN_SCREEN;
END_VAR
VAR_INPUT
	Iin_X : INT;
	Iin_Y : INT;
	Iin_Width : INT;
	Idw_ATTR_1 : DWORD;
	Idw_ATTR_2 : DWORD;
	Iti_TIME : TIME;
END_VAR

(*
version 1.0		10. mai 2010
programmer		ks
tested by		ks

TN_SC_VIEWPORT verwaltet und zeichnet einen rechteckigen Bereich in dem der Log-buffer angezeigt wird
*)
(* LOG-Messages ausgeben *)

IF Xus_LOG_VIEWPORT.UPDATE AND FB_TON.Q THEN (* Update gewünscht und Verzögerungszeit abgelaufen *)
	Xus_LOG_VIEWPORT.UPDATE := FALSE;
	FOR in_count := 1 TO Xus_LOG_VIEWPORT.COUNT DO (* Alle Viewport-Zeilen abarbeiten *)
		in_index := Xus_LOG_VIEWPORT.LINE_ARRAY[in_count];
		(* Farbe aus den Option-Parameter auslesen >0,Level,Back,Front< *)
		in_Color := DWORD_TO_INT(Xus_LOG_CONTROL.MSG_OPTION[in_index] AND DWORD#2#1111);

		CASE in_Color OF
		0..3: by_Attr := BYTE_OF_DWORD(Idw_ATTR_1,INT_TO_BYTE(in_Color));
		4..7: by_Attr := BYTE_OF_DWORD(Idw_ATTR_2,INT_TO_BYTE(in_Color));
		ELSE
			by_Attr := BYTE_OF_DWORD(Idw_ATTR_1,BYTE#0);
		END_CASE;

		(* Message (Text + Farbe) ausgeben *)
		FB_TN_SC_WRITE(	Iin_Y := Iin_Y + in_count - INT#01,
						Iin_X := Iin_X,
						Iby_ATTR := by_Attr,
						Ist_STRING := FIX(str := Xus_LOG_CONTROL.MSG[in_index], L := Iin_Width, C := BYTE#32, M := INT#00), (* String rechts ergänzen bzw. kürzen *)
						Xus_TN_SCREEN := Xus_TN_SCREEN);

	END_FOR;

	(* Timer stoppen/rücksetzen *)
	FB_TON.IN := FALSE;
	FB_TON.PT := Iti_TIME;
	FB_TON();

END_IF;

(* Update-Zeitverzoegerung *)
FB_TON.IN := TRUE;
FB_TON.PT := Iti_TIME;
FB_TON();

(* revision history
ks	10. mai. 2010	rev 1.0
	original version
*)
END_FUNCTION_BLOCK

(* POU TN_VISION_DEMO_2, ST *)
PROGRAM TN_VISION_DEMO_2
VAR
	FB_TN_FRAMEWORK : TN_FRAMEWORK;
	FB_TN_SC_FILL : TN_SC_FILL;
	FB_TN_SC_WRITE_C : TN_SC_WRITE_C;
	FB_TN_SC_WRITE : TN_SC_WRITE;
	Xus_TN_MENU : us_TN_MENU;
	Xus_TN_INPUT_CONTROL : us_TN_INPUT_CONTROL;
	Xus_TN_SCREEN : us_TN_SCREEN;
	S_BUF : NETWORK_BUFFER;
	R_BUF : NETWORK_BUFFER;
	IP_C : IP_C;
END_VAR
FB_TN_FRAMEWORK(
					us_TN_INPUT_CONTROL := Xus_TN_INPUT_CONTROL ,
					us_TN_SCREEN := Xus_TN_SCREEN ,
					us_TN_MENU := Xus_TN_MENU ,
					S_BUF := S_BUF ,
					R_BUF:= R_BUF ,
					IP_C:= IP_C ,
					PORT := WORD#0
					 );


(* Initialisierung der Daten und Strukturen *)
IF (Xus_TN_SCREEN.in_Page_Number = INT#00) THEN
	Xus_TN_SCREEN.in_Page_Number := INT#01;

	(* Clear-Screen (Farbe setzen + Display löschen) *)
	Xus_TN_SCREEN.by_Clear_Screen_Attr := BYTE#16#00;
	Xus_TN_SCREEN.bo_Clear_Screen := TRUE;

	(* Screen initialisieren (mit Leerzeichen füllen) *)
	FB_TN_SC_FILL(	Iin_X1 := INT#00,
					Iin_Y1 := INT#00,
					Iin_X2 := INT#79,
					Iin_Y2 := INT#23,
					Iby_CHAR := BYTE#32,
					Iby_Attr := BYTE#16#00,
					Xus_TN_SCREEN := Xus_TN_SCREEN);

	(* Statische Texte ausgeben *)
	FB_TN_SC_WRITE(	Iin_X := INT#00,
					Iin_Y := INT#00,
					Iby_ATTR := BYTE#16#70,
					Ist_STRING := 'Login Screen                                                     FL SWITCH MM HS',
					Xus_TN_SCREEN := Xus_TN_SCREEN);

	(* Statische Texte ausgeben *)
	FB_TN_SC_WRITE(	Iin_X := INT#00,
					Iin_Y := INT#03,
					Iby_ATTR := BYTE#16#70,
					Ist_STRING := 'XXXXXXXXX',
					Xus_TN_SCREEN := Xus_TN_SCREEN);

	(* Statische Texte ausgeben *)
	FB_TN_SC_WRITE(	Iin_X := INT#00,
					Iin_Y := INT#04,
					Iby_ATTR := BYTE#16#70,
					Ist_STRING := 'X   X  XX',
					Xus_TN_SCREEN := Xus_TN_SCREEN);

	(* Statische Texte ausgeben *)
	FB_TN_SC_WRITE(	Iin_X := INT#00,
					Iin_Y := INT#05,
					Iby_ATTR := BYTE#16#70,
					Ist_STRING := 'X   O   X      ---> Phoenix Contact Managed Switch System <---',
					Xus_TN_SCREEN := Xus_TN_SCREEN);

	(* Statische Texte ausgeben *)
	FB_TN_SC_WRITE(	Iin_X := INT#00,
					Iin_Y := INT#06,
					Iby_ATTR := BYTE#16#70,
					Ist_STRING := 'X   X  XX               Phoenix Contact GmbH & Co KG',
					Xus_TN_SCREEN := Xus_TN_SCREEN);

	(* Statische Texte ausgeben *)
	FB_TN_SC_WRITE(	Iin_X := INT#00,
					Iin_Y := INT#07,
					Iby_ATTR := BYTE#16#70,
					Ist_STRING := 'X   XXXXX                   www.PhoenixContact.com',
					Xus_TN_SCREEN := Xus_TN_SCREEN);

	(* Statische Texte ausgeben *)
	FB_TN_SC_WRITE(	Iin_X := INT#00,
					Iin_Y := INT#08,
					Iby_ATTR := BYTE#16#70,
					Ist_STRING := 'X   XXXXX',
					Xus_TN_SCREEN := Xus_TN_SCREEN);

	(* Statische Texte ausgeben *)
	FB_TN_SC_WRITE(	Iin_X := INT#00,
					Iin_Y := INT#09,
					Iby_ATTR := BYTE#16#70,
					Ist_STRING := 'XXXXXXXXX',
					Xus_TN_SCREEN := Xus_TN_SCREEN);

	(* Statische Texte ausgeben *)
	FB_TN_SC_WRITE(	Iin_X := INT#00,
					Iin_Y := INT#11,
					Iby_ATTR := BYTE#16#70,
					Ist_STRING := '                Running switch application version:  4.00',
					Xus_TN_SCREEN := Xus_TN_SCREEN);

	(* Alle Input-Controls initialisieren *)

	Xus_TN_INPUT_CONTROL.bo_Enable := FALSE;

  (* Initialisierung der Eingabe-Zeile *)
	Xus_TN_INPUT_CONTROL.usa_TN_INPUT_CONTROL_DATA[1].in_Type := INT#01;
	Xus_TN_INPUT_CONTROL.usa_TN_INPUT_CONTROL_DATA[1].in_Y := INT#17;
	Xus_TN_INPUT_CONTROL.usa_TN_INPUT_CONTROL_DATA[1].in_X := INT#33;
	Xus_TN_INPUT_CONTROL.usa_TN_INPUT_CONTROL_DATA[1].by_Attr_mF := BYTE#16#70;
	Xus_TN_INPUT_CONTROL.usa_TN_INPUT_CONTROL_DATA[1].by_Attr_oF := BYTE#16#70;
	Xus_TN_INPUT_CONTROL.usa_TN_INPUT_CONTROL_DATA[1].in_Cursor_Pos := INT#0;
	Xus_TN_INPUT_CONTROL.usa_TN_INPUT_CONTROL_DATA[1].bo_Input_Only_Num := FALSE;
	Xus_TN_INPUT_CONTROL.usa_TN_INPUT_CONTROL_DATA[1].bo_Input_Hidden := TRUE;
	Xus_TN_INPUT_CONTROL.usa_TN_INPUT_CONTROL_DATA[1].st_Input_Mask := '                ';
	Xus_TN_INPUT_CONTROL.usa_TN_INPUT_CONTROL_DATA[1].st_Input_Data := Xus_TN_INPUT_CONTROL.usa_TN_INPUT_CONTROL_DATA[1].st_Input_Mask;
	Xus_TN_INPUT_CONTROL.usa_TN_INPUT_CONTROL_DATA[1].st_Input_ToolTip := '';
	Xus_TN_INPUT_CONTROL.usa_TN_INPUT_CONTROL_DATA[1].in_Input_Option := INT#00;
	Xus_TN_INPUT_CONTROL.usa_TN_INPUT_CONTROL_DATA[1].in_Title_Y_Offset := INT#00;
	Xus_TN_INPUT_CONTROL.usa_TN_INPUT_CONTROL_DATA[1].in_Title_X_Offset := -12;
	Xus_TN_INPUT_CONTROL.usa_TN_INPUT_CONTROL_DATA[1].by_Title_Attr := BYTE#16#70;
	Xus_TN_INPUT_CONTROL.usa_TN_INPUT_CONTROL_DATA[1].st_Title_String := 'Password:  [                ]';

	(* Control-Tool-Tip *)
	Xus_TN_INPUT_CONTROL.in_ToolTip_Y := INT#23;
	Xus_TN_INPUT_CONTROL.in_ToolTip_X := INT#09;
	Xus_TN_INPUT_CONTROL.by_ToolTip_Attr := BYTE#16#70;
	Xus_TN_INPUT_CONTROL.in_ToolTip_Size := INT#30;

	(* Control-Verwaltung initialisieren *)
	Xus_TN_INPUT_CONTROL.in_Count := INT#01;
	Xus_TN_INPUT_CONTROL.bo_Enable := TRUE;
	Xus_TN_INPUT_CONTROL.bo_Reset_Fokus := TRUE;
END_IF;

IF (Xus_TN_SCREEN.in_Page_Number = INT#01) THEN

	(* eingegebenen String übernehmen *)
	IF Xus_TN_INPUT_CONTROL.usa_TN_INPUT_CONTROL_DATA[1].bo_Input_Entered = TRUE THEN

		Xus_TN_INPUT_CONTROL.usa_TN_INPUT_CONTROL_DATA[1].bo_Input_Entered := FALSE;

		Xus_TN_INPUT_CONTROL.usa_TN_INPUT_CONTROL_DATA[1].st_Input_String :=
			LOWERCASE(str:=Xus_TN_INPUT_CONTROL.usa_TN_INPUT_CONTROL_DATA[1].st_Input_String);

		IF Xus_TN_INPUT_CONTROL.usa_TN_INPUT_CONTROL_DATA[1].st_Input_String = 'oscat' THEN
			Xus_TN_SCREEN.in_Page_Number := INT#04;

		ELSE
			FB_TN_SC_WRITE_C(	Iin_Y := Xus_TN_INPUT_CONTROL.in_ToolTip_Y,
								Iin_X := Xus_TN_INPUT_CONTROL.in_ToolTip_X,
								Iby_ATTR := BYTE#16#F1,
								Iin_OPTION := INT#02, (* Center-String *)
								Iin_LENGTH := Xus_TN_INPUT_CONTROL.in_ToolTip_Size,
								Ist_STRING := ' User Password Failed   ',
								Xus_TN_SCREEN := Xus_TN_SCREEN);
		END_IF;
	END_IF;
END_IF;

(* Initialisierung der Daten und Strukturen *)
IF (Xus_TN_SCREEN.in_Page_Number = INT#04) THEN
	Xus_TN_SCREEN.in_Page_Number := INT#05;

	(* Clear-Screen (Farbe setzen + Display löschen) *)
	Xus_TN_SCREEN.by_Clear_Screen_Attr := BYTE#16#00;
	Xus_TN_SCREEN.bo_Clear_Screen := TRUE;

	(* Screen initialisieren (mit Leerzeichen füllen) *)
	FB_TN_SC_FILL(	Iin_X1 := INT#00,
					Iin_Y1 := INT#00,
					Iin_X2 := INT#79,
					Iin_Y2 := INT#23,
					Iby_CHAR := BYTE#32,
					Iby_Attr := BYTE#16#00,
					Xus_TN_SCREEN := Xus_TN_SCREEN);

	(* Statische Texte ausgeben *)
	FB_TN_SC_WRITE(	Iin_X := INT#00,
					Iin_Y := INT#00,
					Iby_ATTR := BYTE#16#70,
					Ist_STRING := 'Basic Switch Configuration                                       FL SWITCH MM HS',
					Xus_TN_SCREEN := Xus_TN_SCREEN);

	(* Statische Texte ausgeben                                         *)
	FB_TN_SC_WRITE(	Iin_X := INT#00,
					Iin_Y := INT#03,
					Iby_ATTR := BYTE#16#70,
					Ist_STRING := 'XXXXXXXXX        MAC Address             : 00:A0:45:00:6E:9B',
					Xus_TN_SCREEN := Xus_TN_SCREEN);

	(* Statische Texte ausgeben *)
	FB_TN_SC_WRITE(	Iin_X := INT#00,
					Iin_Y := INT#04,
					Iby_ATTR := BYTE#16#70,
					Ist_STRING := 'X   X  XX',
					Xus_TN_SCREEN := Xus_TN_SCREEN);

	(* Statische Texte ausgeben *)
	FB_TN_SC_WRITE(	Iin_X := INT#00,
					Iin_Y := INT#05,
					Iby_ATTR := BYTE#16#70,
					Ist_STRING := 'X   O   X',
					Xus_TN_SCREEN := Xus_TN_SCREEN);

	(* Statische Texte ausgeben *)
	FB_TN_SC_WRITE(	Iin_X := INT#00,
					Iin_Y := INT#06,
					Iby_ATTR := BYTE#16#70,
					Ist_STRING := 'X   X  XX',
					Xus_TN_SCREEN := Xus_TN_SCREEN);

	(* Statische Texte ausgeben *)
	FB_TN_SC_WRITE(	Iin_X := INT#00,
					Iin_Y := INT#07,
					Iby_ATTR := BYTE#16#70,
					Ist_STRING := 'X   XXXXX',
					Xus_TN_SCREEN := Xus_TN_SCREEN);

	(* Statische Texte ausgeben *)
	FB_TN_SC_WRITE(	Iin_X := INT#00,
					Iin_Y := INT#08,
					Iby_ATTR := BYTE#16#70,
					Ist_STRING := 'X   XXXXX',
					Xus_TN_SCREEN := Xus_TN_SCREEN);

	(* Statische Texte ausgeben *)
	FB_TN_SC_WRITE(	Iin_X := INT#00,
					Iin_Y := INT#09,
					Iby_ATTR := BYTE#16#70,
					Ist_STRING := 'XXXXXXXXX',
					Xus_TN_SCREEN := Xus_TN_SCREEN);

	(* Alle Input-Controls initialisieren *)

	Xus_TN_INPUT_CONTROL.bo_Enable      := FALSE;

	Xus_TN_INPUT_CONTROL.usa_TN_INPUT_CONTROL_DATA[1].in_Type := INT#01;
	Xus_TN_INPUT_CONTROL.usa_TN_INPUT_CONTROL_DATA[1].in_Y := INT#04;
	Xus_TN_INPUT_CONTROL.usa_TN_INPUT_CONTROL_DATA[1].in_X := INT#44;
	Xus_TN_INPUT_CONTROL.usa_TN_INPUT_CONTROL_DATA[1].by_Attr_mF := BYTE#16#07; (* Weiss, Grün *)
	Xus_TN_INPUT_CONTROL.usa_TN_INPUT_CONTROL_DATA[1].by_Attr_oF := BYTE#16#70; (* Weiss, Blau *)
	Xus_TN_INPUT_CONTROL.usa_TN_INPUT_CONTROL_DATA[1].in_Cursor_Pos := INT#0;
	Xus_TN_INPUT_CONTROL.usa_TN_INPUT_CONTROL_DATA[1].bo_Input_Only_Num := TRUE;
	Xus_TN_INPUT_CONTROL.usa_TN_INPUT_CONTROL_DATA[1].bo_Input_Hidden := FALSE;
	Xus_TN_INPUT_CONTROL.usa_TN_INPUT_CONTROL_DATA[1].st_Input_Mask := '   .   .   .   ';
	Xus_TN_INPUT_CONTROL.usa_TN_INPUT_CONTROL_DATA[1].st_Input_Data := Xus_TN_INPUT_CONTROL.usa_TN_INPUT_CONTROL_DATA[1].st_Input_Mask;
	Xus_TN_INPUT_CONTROL.usa_TN_INPUT_CONTROL_DATA[1].st_Input_ToolTip := 'Enter Agent IP Address in decimal dot format (e.g., 209.131.209.13)';
	Xus_TN_INPUT_CONTROL.usa_TN_INPUT_CONTROL_DATA[1].in_Input_Option := INT#01;
	Xus_TN_INPUT_CONTROL.usa_TN_INPUT_CONTROL_DATA[1].in_Title_Y_Offset := INT#00;
	Xus_TN_INPUT_CONTROL.usa_TN_INPUT_CONTROL_DATA[1].in_Title_X_Offset := -27;
	Xus_TN_INPUT_CONTROL.usa_TN_INPUT_CONTROL_DATA[1].by_Title_Attr := BYTE#16#70;
	Xus_TN_INPUT_CONTROL.usa_TN_INPUT_CONTROL_DATA[1].st_Title_String := 'IP Address              : [149.208.100.100]';

	Xus_TN_INPUT_CONTROL.usa_TN_INPUT_CONTROL_DATA[2].in_Type := INT#01;
	Xus_TN_INPUT_CONTROL.usa_TN_INPUT_CONTROL_DATA[2].in_Y := INT#05;
	Xus_TN_INPUT_CONTROL.usa_TN_INPUT_CONTROL_DATA[2].in_X := INT#44;
	Xus_TN_INPUT_CONTROL.usa_TN_INPUT_CONTROL_DATA[2].by_Attr_mF := BYTE#16#07; (* Weiss, Grün *)
	Xus_TN_INPUT_CONTROL.usa_TN_INPUT_CONTROL_DATA[2].by_Attr_oF := BYTE#16#70; (* Weiss, Blau *)
	Xus_TN_INPUT_CONTROL.usa_TN_INPUT_CONTROL_DATA[2].in_Cursor_Pos := INT#0;
	Xus_TN_INPUT_CONTROL.usa_TN_INPUT_CONTROL_DATA[2].bo_Input_Only_Num := TRUE;
	Xus_TN_INPUT_CONTROL.usa_TN_INPUT_CONTROL_DATA[2].bo_Input_Hidden := FALSE;
	Xus_TN_INPUT_CONTROL.usa_TN_INPUT_CONTROL_DATA[2].st_Input_Mask := '   .   .   .   ';
	Xus_TN_INPUT_CONTROL.usa_TN_INPUT_CONTROL_DATA[2].st_Input_Data := Xus_TN_INPUT_CONTROL.usa_TN_INPUT_CONTROL_DATA[1].st_Input_Mask;
	Xus_TN_INPUT_CONTROL.usa_TN_INPUT_CONTROL_DATA[2].st_Input_ToolTip := 'Enter Agent Netmask (e.g., 255.255.255.0)';
	Xus_TN_INPUT_CONTROL.usa_TN_INPUT_CONTROL_DATA[2].in_Input_Option := INT#01;
	Xus_TN_INPUT_CONTROL.usa_TN_INPUT_CONTROL_DATA[2].in_Title_Y_Offset := INT#00;
	Xus_TN_INPUT_CONTROL.usa_TN_INPUT_CONTROL_DATA[2].in_Title_X_Offset := -27;
	Xus_TN_INPUT_CONTROL.usa_TN_INPUT_CONTROL_DATA[2].by_Title_Attr := BYTE#16#70;
	Xus_TN_INPUT_CONTROL.usa_TN_INPUT_CONTROL_DATA[2].st_Title_String := 'Subnet Mask             : [255.255.255.128]';

	Xus_TN_INPUT_CONTROL.usa_TN_INPUT_CONTROL_DATA[3].in_Type := INT#01;
	Xus_TN_INPUT_CONTROL.usa_TN_INPUT_CONTROL_DATA[3].in_Y := INT#06;
	Xus_TN_INPUT_CONTROL.usa_TN_INPUT_CONTROL_DATA[3].in_X := INT#44;
	Xus_TN_INPUT_CONTROL.usa_TN_INPUT_CONTROL_DATA[3].by_Attr_mF := BYTE#16#07; (* Weiss, Grün *)
	Xus_TN_INPUT_CONTROL.usa_TN_INPUT_CONTROL_DATA[3].by_Attr_oF := BYTE#16#70; (* Weiss, Blau *)
	Xus_TN_INPUT_CONTROL.usa_TN_INPUT_CONTROL_DATA[3].in_Cursor_Pos := INT#0;
	Xus_TN_INPUT_CONTROL.usa_TN_INPUT_CONTROL_DATA[3].bo_Input_Only_Num := TRUE;
	Xus_TN_INPUT_CONTROL.usa_TN_INPUT_CONTROL_DATA[3].bo_Input_Hidden := FALSE;
	Xus_TN_INPUT_CONTROL.usa_TN_INPUT_CONTROL_DATA[3].st_Input_Mask := '   .   .   .   ';
	Xus_TN_INPUT_CONTROL.usa_TN_INPUT_CONTROL_DATA[3].st_Input_Data := Xus_TN_INPUT_CONTROL.usa_TN_INPUT_CONTROL_DATA[1].st_Input_Mask;
	Xus_TN_INPUT_CONTROL.usa_TN_INPUT_CONTROL_DATA[3].st_Input_ToolTip := 'Enter Agent Default Gateway, (e.g., 209.131.209.1)';
	Xus_TN_INPUT_CONTROL.usa_TN_INPUT_CONTROL_DATA[3].in_Input_Option := INT#01;
	Xus_TN_INPUT_CONTROL.usa_TN_INPUT_CONTROL_DATA[3].in_Title_Y_Offset := INT#00;
	Xus_TN_INPUT_CONTROL.usa_TN_INPUT_CONTROL_DATA[3].in_Title_X_Offset := -27;
	Xus_TN_INPUT_CONTROL.usa_TN_INPUT_CONTROL_DATA[3].by_Title_Attr := BYTE#16#70;
	Xus_TN_INPUT_CONTROL.usa_TN_INPUT_CONTROL_DATA[3].st_Title_String := 'Default Gateway         : [149.208.100.1  ]';

	Xus_TN_INPUT_CONTROL.usa_TN_INPUT_CONTROL_DATA[4].in_Type := INT#02;
	Xus_TN_INPUT_CONTROL.usa_TN_INPUT_CONTROL_DATA[4].in_Y := INT#07;
	Xus_TN_INPUT_CONTROL.usa_TN_INPUT_CONTROL_DATA[4].in_X := INT#44;
	Xus_TN_INPUT_CONTROL.usa_TN_INPUT_CONTROL_DATA[4].by_Attr_mF := BYTE#16#07;
	Xus_TN_INPUT_CONTROL.usa_TN_INPUT_CONTROL_DATA[4].by_Attr_oF := BYTE#16#70;
	Xus_TN_INPUT_CONTROL.usa_TN_INPUT_CONTROL_DATA[4].st_Input_Mask := '       ';
	Xus_TN_INPUT_CONTROL.usa_TN_INPUT_CONTROL_DATA[4].st_Input_Data := 'BootP  #DHCP   #DCP    #Static ';
	Xus_TN_INPUT_CONTROL.usa_TN_INPUT_CONTROL_DATA[4].st_Input_ToolTip := 'Push SPACE to select the address assignment (effective after reboot)';
	Xus_TN_INPUT_CONTROL.usa_TN_INPUT_CONTROL_DATA[4].in_Input_Option := INT#02;
	Xus_TN_INPUT_CONTROL.usa_TN_INPUT_CONTROL_DATA[4].in_Title_Y_Offset := INT#00;
	Xus_TN_INPUT_CONTROL.usa_TN_INPUT_CONTROL_DATA[4].in_Title_X_Offset := -27;
	Xus_TN_INPUT_CONTROL.usa_TN_INPUT_CONTROL_DATA[4].by_Title_Attr := BYTE#16#70;
	Xus_TN_INPUT_CONTROL.usa_TN_INPUT_CONTROL_DATA[4].st_Title_String := 'IP Parameter Assignment : <BootP  >';

	Xus_TN_INPUT_CONTROL.usa_TN_INPUT_CONTROL_DATA[5].in_Type := INT#02;
	Xus_TN_INPUT_CONTROL.usa_TN_INPUT_CONTROL_DATA[5].in_Y := INT#09;
	Xus_TN_INPUT_CONTROL.usa_TN_INPUT_CONTROL_DATA[5].in_X := INT#44;
	Xus_TN_INPUT_CONTROL.usa_TN_INPUT_CONTROL_DATA[5].by_Attr_mF := BYTE#16#07;
	Xus_TN_INPUT_CONTROL.usa_TN_INPUT_CONTROL_DATA[5].by_Attr_oF := BYTE#16#70;
	Xus_TN_INPUT_CONTROL.usa_TN_INPUT_CONTROL_DATA[5].st_Input_Mask := '                              ';
	Xus_TN_INPUT_CONTROL.usa_TN_INPUT_CONTROL_DATA[5].st_Input_Data := 'No Redundancy#Rapid Spanning Tree, Disabled#Rapid Spanning Tree, Enabled';
	Xus_TN_INPUT_CONTROL.usa_TN_INPUT_CONTROL_DATA[5].st_Input_ToolTip := 'Push SPACE to chose redundancy (network disruption for few seconds if enabled)';
	Xus_TN_INPUT_CONTROL.usa_TN_INPUT_CONTROL_DATA[5].in_Input_Option := INT#02;
	Xus_TN_INPUT_CONTROL.usa_TN_INPUT_CONTROL_DATA[5].in_Title_Y_Offset := INT#00;
	Xus_TN_INPUT_CONTROL.usa_TN_INPUT_CONTROL_DATA[5].in_Title_X_Offset := -27;
	Xus_TN_INPUT_CONTROL.usa_TN_INPUT_CONTROL_DATA[5].by_Title_Attr := BYTE#16#70;
	Xus_TN_INPUT_CONTROL.usa_TN_INPUT_CONTROL_DATA[5].st_Title_String := 'Redundancy              : <No Redundancy                 >';

	(* Statische Texte ausgeben *)
	FB_TN_SC_WRITE(	Iin_X := INT#17,
					Iin_Y := INT#10,
					Iby_ATTR := BYTE#16#70,
					Ist_STRING := 'Current Vlan Status     :  VLAN Transparent',
					Xus_TN_SCREEN := Xus_TN_SCREEN);

	Xus_TN_INPUT_CONTROL.usa_TN_INPUT_CONTROL_DATA[6].in_Type := INT#02;
	Xus_TN_INPUT_CONTROL.usa_TN_INPUT_CONTROL_DATA[6].in_Y := INT#11;
	Xus_TN_INPUT_CONTROL.usa_TN_INPUT_CONTROL_DATA[6].in_X := INT#44;
	Xus_TN_INPUT_CONTROL.usa_TN_INPUT_CONTROL_DATA[6].by_Attr_mF := BYTE#16#07;
	Xus_TN_INPUT_CONTROL.usa_TN_INPUT_CONTROL_DATA[6].by_Attr_oF := BYTE#16#70;
	Xus_TN_INPUT_CONTROL.usa_TN_INPUT_CONTROL_DATA[6].st_Input_Mask := '                        ';
	Xus_TN_INPUT_CONTROL.usa_TN_INPUT_CONTROL_DATA[6].st_Input_Data := 'VLAN Transparent#VLAN Tagging';
	Xus_TN_INPUT_CONTROL.usa_TN_INPUT_CONTROL_DATA[6].st_Input_ToolTip := 'Push SPACE to toggle the VLAN Mode (effective after reboot)';
	Xus_TN_INPUT_CONTROL.usa_TN_INPUT_CONTROL_DATA[6].in_Input_Option := INT#02;
	Xus_TN_INPUT_CONTROL.usa_TN_INPUT_CONTROL_DATA[6].in_Title_Y_Offset := INT#00;
	Xus_TN_INPUT_CONTROL.usa_TN_INPUT_CONTROL_DATA[6].in_Title_X_Offset := -27;
	Xus_TN_INPUT_CONTROL.usa_TN_INPUT_CONTROL_DATA[6].by_Title_Attr := BYTE#16#70;
	Xus_TN_INPUT_CONTROL.usa_TN_INPUT_CONTROL_DATA[6].st_Title_String := 'Vlan Mode               : <VLAN Transparent        >';

	Xus_TN_INPUT_CONTROL.usa_TN_INPUT_CONTROL_DATA[7].in_Type := INT#02;
	Xus_TN_INPUT_CONTROL.usa_TN_INPUT_CONTROL_DATA[7].in_Y := INT#12;
	Xus_TN_INPUT_CONTROL.usa_TN_INPUT_CONTROL_DATA[7].in_X := INT#44;
	Xus_TN_INPUT_CONTROL.usa_TN_INPUT_CONTROL_DATA[7].by_Attr_mF := BYTE#16#07;
	Xus_TN_INPUT_CONTROL.usa_TN_INPUT_CONTROL_DATA[7].by_Attr_oF := BYTE#16#70;
	Xus_TN_INPUT_CONTROL.usa_TN_INPUT_CONTROL_DATA[7].st_Input_Mask := '       ';
	Xus_TN_INPUT_CONTROL.usa_TN_INPUT_CONTROL_DATA[7].st_Input_Data := 'Disable#Enable';
	Xus_TN_INPUT_CONTROL.usa_TN_INPUT_CONTROL_DATA[7].st_Input_ToolTip := 'Push SPACE to Enable/Disable Port Security';
	Xus_TN_INPUT_CONTROL.usa_TN_INPUT_CONTROL_DATA[7].in_Input_Option := INT#02;
	Xus_TN_INPUT_CONTROL.usa_TN_INPUT_CONTROL_DATA[7].in_Title_Y_Offset := INT#00;
	Xus_TN_INPUT_CONTROL.usa_TN_INPUT_CONTROL_DATA[7].in_Title_X_Offset := -27;
	Xus_TN_INPUT_CONTROL.usa_TN_INPUT_CONTROL_DATA[7].by_Title_Attr := BYTE#16#70;
	Xus_TN_INPUT_CONTROL.usa_TN_INPUT_CONTROL_DATA[7].st_Title_String := 'Port Security           : <Disable>';

	Xus_TN_INPUT_CONTROL.usa_TN_INPUT_CONTROL_DATA[8].in_Type := INT#02;
	Xus_TN_INPUT_CONTROL.usa_TN_INPUT_CONTROL_DATA[8].in_Y := INT#13;
	Xus_TN_INPUT_CONTROL.usa_TN_INPUT_CONTROL_DATA[8].in_X := INT#44;
	Xus_TN_INPUT_CONTROL.usa_TN_INPUT_CONTROL_DATA[8].by_Attr_mF := BYTE#16#07;
	Xus_TN_INPUT_CONTROL.usa_TN_INPUT_CONTROL_DATA[8].by_Attr_oF := BYTE#16#70;
	Xus_TN_INPUT_CONTROL.usa_TN_INPUT_CONTROL_DATA[8].st_Input_Mask := '       ';
	Xus_TN_INPUT_CONTROL.usa_TN_INPUT_CONTROL_DATA[8].st_Input_Data := 'Disable#Enable';
	Xus_TN_INPUT_CONTROL.usa_TN_INPUT_CONTROL_DATA[8].st_Input_ToolTip := 'Push SPACE to Enable/Disable Access Control for the WEB Interface';
	Xus_TN_INPUT_CONTROL.usa_TN_INPUT_CONTROL_DATA[8].in_Input_Option := INT#02;
	Xus_TN_INPUT_CONTROL.usa_TN_INPUT_CONTROL_DATA[8].in_Title_Y_Offset := INT#00;
	Xus_TN_INPUT_CONTROL.usa_TN_INPUT_CONTROL_DATA[8].in_Title_X_Offset := -27;
	Xus_TN_INPUT_CONTROL.usa_TN_INPUT_CONTROL_DATA[8].by_Title_Attr := BYTE#16#70;
	Xus_TN_INPUT_CONTROL.usa_TN_INPUT_CONTROL_DATA[8].st_Title_String := 'Access Control for Web  : <Disable>';

	Xus_TN_INPUT_CONTROL.usa_TN_INPUT_CONTROL_DATA[9].in_Type := INT#02;
	Xus_TN_INPUT_CONTROL.usa_TN_INPUT_CONTROL_DATA[9].in_Y := INT#14;
	Xus_TN_INPUT_CONTROL.usa_TN_INPUT_CONTROL_DATA[9].in_X := INT#44;
	Xus_TN_INPUT_CONTROL.usa_TN_INPUT_CONTROL_DATA[9].by_Attr_mF := BYTE#16#07;
	Xus_TN_INPUT_CONTROL.usa_TN_INPUT_CONTROL_DATA[9].by_Attr_oF := BYTE#16#70;
	Xus_TN_INPUT_CONTROL.usa_TN_INPUT_CONTROL_DATA[9].st_Input_Mask := '        ';
	Xus_TN_INPUT_CONTROL.usa_TN_INPUT_CONTROL_DATA[9].st_Input_Data := 'Default#Profinet';
	Xus_TN_INPUT_CONTROL.usa_TN_INPUT_CONTROL_DATA[9].st_Input_ToolTip := 'Push SPACE to select the switch operating mode';
	Xus_TN_INPUT_CONTROL.usa_TN_INPUT_CONTROL_DATA[9].in_Input_Option := INT#02;
	Xus_TN_INPUT_CONTROL.usa_TN_INPUT_CONTROL_DATA[9].in_Title_Y_Offset := INT#00;
	Xus_TN_INPUT_CONTROL.usa_TN_INPUT_CONTROL_DATA[9].in_Title_X_Offset := -27;
	Xus_TN_INPUT_CONTROL.usa_TN_INPUT_CONTROL_DATA[9].by_Title_Attr := BYTE#16#70;
	Xus_TN_INPUT_CONTROL.usa_TN_INPUT_CONTROL_DATA[9].st_Title_String := 'Switch Operating Mode   : <Default >';

	Xus_TN_INPUT_CONTROL.usa_TN_INPUT_CONTROL_DATA[10].in_Type := INT#02;
	Xus_TN_INPUT_CONTROL.usa_TN_INPUT_CONTROL_DATA[10].in_Y := INT#16;
	Xus_TN_INPUT_CONTROL.usa_TN_INPUT_CONTROL_DATA[10].in_X := INT#44;
	Xus_TN_INPUT_CONTROL.usa_TN_INPUT_CONTROL_DATA[10].by_Attr_mF := BYTE#16#07;
	Xus_TN_INPUT_CONTROL.usa_TN_INPUT_CONTROL_DATA[10].by_Attr_oF := BYTE#16#70;
	Xus_TN_INPUT_CONTROL.usa_TN_INPUT_CONTROL_DATA[10].st_Input_Mask := '       ';
	Xus_TN_INPUT_CONTROL.usa_TN_INPUT_CONTROL_DATA[10].st_Input_Data := 'Enable#Disable';
	Xus_TN_INPUT_CONTROL.usa_TN_INPUT_CONTROL_DATA[10].st_Input_ToolTip := 'Push SPACE to Enable/Disable Web Interface (effective after reboot)';
	Xus_TN_INPUT_CONTROL.usa_TN_INPUT_CONTROL_DATA[10].in_Input_Option := INT#02;
	Xus_TN_INPUT_CONTROL.usa_TN_INPUT_CONTROL_DATA[10].in_Title_Y_Offset := INT#00;
	Xus_TN_INPUT_CONTROL.usa_TN_INPUT_CONTROL_DATA[10].in_Title_X_Offset := -27;
	Xus_TN_INPUT_CONTROL.usa_TN_INPUT_CONTROL_DATA[10].by_Title_Attr := BYTE#16#70;
	Xus_TN_INPUT_CONTROL.usa_TN_INPUT_CONTROL_DATA[10].st_Title_String := 'Web Interface           : <Enable >';

	Xus_TN_INPUT_CONTROL.usa_TN_INPUT_CONTROL_DATA[11].in_Type := INT#02;
	Xus_TN_INPUT_CONTROL.usa_TN_INPUT_CONTROL_DATA[11].in_Y := INT#17;
	Xus_TN_INPUT_CONTROL.usa_TN_INPUT_CONTROL_DATA[11].in_X := INT#44;
	Xus_TN_INPUT_CONTROL.usa_TN_INPUT_CONTROL_DATA[11].by_Attr_mF := BYTE#16#07;
	Xus_TN_INPUT_CONTROL.usa_TN_INPUT_CONTROL_DATA[11].by_Attr_oF := BYTE#16#70;
	Xus_TN_INPUT_CONTROL.usa_TN_INPUT_CONTROL_DATA[11].st_Input_Mask := '       ';
	Xus_TN_INPUT_CONTROL.usa_TN_INPUT_CONTROL_DATA[11].st_Input_Data := 'Enable#Disable';
	Xus_TN_INPUT_CONTROL.usa_TN_INPUT_CONTROL_DATA[11].st_Input_ToolTip := 'Push SPACE to Enable/Disable Telnet Interface (effective after reboot)';
	Xus_TN_INPUT_CONTROL.usa_TN_INPUT_CONTROL_DATA[11].in_Input_Option := INT#02;
	Xus_TN_INPUT_CONTROL.usa_TN_INPUT_CONTROL_DATA[11].in_Title_Y_Offset := INT#00;
	Xus_TN_INPUT_CONTROL.usa_TN_INPUT_CONTROL_DATA[11].in_Title_X_Offset := -27;
	Xus_TN_INPUT_CONTROL.usa_TN_INPUT_CONTROL_DATA[11].by_Title_Attr := BYTE#16#70;
	Xus_TN_INPUT_CONTROL.usa_TN_INPUT_CONTROL_DATA[11].st_Title_String := 'Telnet Interface        : <Enable >';

	Xus_TN_INPUT_CONTROL.usa_TN_INPUT_CONTROL_DATA[12].in_Type := INT#02;
	Xus_TN_INPUT_CONTROL.usa_TN_INPUT_CONTROL_DATA[12].in_Y := INT#18;
	Xus_TN_INPUT_CONTROL.usa_TN_INPUT_CONTROL_DATA[12].in_X := INT#44;
	Xus_TN_INPUT_CONTROL.usa_TN_INPUT_CONTROL_DATA[12].by_Attr_mF := BYTE#16#07;
	Xus_TN_INPUT_CONTROL.usa_TN_INPUT_CONTROL_DATA[12].by_Attr_oF := BYTE#16#70;
	Xus_TN_INPUT_CONTROL.usa_TN_INPUT_CONTROL_DATA[12].st_Input_Mask := '       ';
	Xus_TN_INPUT_CONTROL.usa_TN_INPUT_CONTROL_DATA[12].st_Input_Data := 'Enable#Disable';
	Xus_TN_INPUT_CONTROL.usa_TN_INPUT_CONTROL_DATA[12].st_Input_ToolTip := 'Push SPACE to Enable/Disable SNMP Interface (effective after reboot)';
	Xus_TN_INPUT_CONTROL.usa_TN_INPUT_CONTROL_DATA[12].in_Input_Option := INT#02;
	Xus_TN_INPUT_CONTROL.usa_TN_INPUT_CONTROL_DATA[12].in_Title_Y_Offset := INT#00;
	Xus_TN_INPUT_CONTROL.usa_TN_INPUT_CONTROL_DATA[12].in_Title_X_Offset := -27;
	Xus_TN_INPUT_CONTROL.usa_TN_INPUT_CONTROL_DATA[12].by_Title_Attr := BYTE#16#70;
	Xus_TN_INPUT_CONTROL.usa_TN_INPUT_CONTROL_DATA[12].st_Title_String := 'SNMP Interface          : <Enable >';

	Xus_TN_INPUT_CONTROL.usa_TN_INPUT_CONTROL_DATA[13].in_Type := INT#02;
	Xus_TN_INPUT_CONTROL.usa_TN_INPUT_CONTROL_DATA[13].in_Y := INT#20;
	Xus_TN_INPUT_CONTROL.usa_TN_INPUT_CONTROL_DATA[13].in_X := INT#44;
	Xus_TN_INPUT_CONTROL.usa_TN_INPUT_CONTROL_DATA[13].by_Attr_mF := BYTE#16#07;
	Xus_TN_INPUT_CONTROL.usa_TN_INPUT_CONTROL_DATA[13].by_Attr_oF := BYTE#16#70;
	Xus_TN_INPUT_CONTROL.usa_TN_INPUT_CONTROL_DATA[13].st_Input_Mask := '                                 ';
	Xus_TN_INPUT_CONTROL.usa_TN_INPUT_CONTROL_DATA[13].st_Input_Data := 'No reset#Reset Switch#Reset Switch to factory defaults';
	Xus_TN_INPUT_CONTROL.usa_TN_INPUT_CONTROL_DATA[13].st_Input_ToolTip := 'Push SPACE to select Reset Option';
	Xus_TN_INPUT_CONTROL.usa_TN_INPUT_CONTROL_DATA[13].in_Input_Option := INT#02;
	Xus_TN_INPUT_CONTROL.usa_TN_INPUT_CONTROL_DATA[13].in_Title_Y_Offset := INT#00;
	Xus_TN_INPUT_CONTROL.usa_TN_INPUT_CONTROL_DATA[13].in_Title_X_Offset := -27;
	Xus_TN_INPUT_CONTROL.usa_TN_INPUT_CONTROL_DATA[13].by_Title_Attr := BYTE#16#70;
	Xus_TN_INPUT_CONTROL.usa_TN_INPUT_CONTROL_DATA[13].st_Title_String := 'Reset                   : <No reset                         >';

	Xus_TN_INPUT_CONTROL.usa_TN_INPUT_CONTROL_DATA[14].in_Type := INT#02;
	Xus_TN_INPUT_CONTROL.usa_TN_INPUT_CONTROL_DATA[14].in_Y := INT#22;
	Xus_TN_INPUT_CONTROL.usa_TN_INPUT_CONTROL_DATA[14].in_X := INT#18;
	Xus_TN_INPUT_CONTROL.usa_TN_INPUT_CONTROL_DATA[14].by_Attr_mF := BYTE#16#07;
	Xus_TN_INPUT_CONTROL.usa_TN_INPUT_CONTROL_DATA[14].by_Attr_oF := BYTE#16#70;
	Xus_TN_INPUT_CONTROL.usa_TN_INPUT_CONTROL_DATA[14].st_Input_ToolTip := 'Apply and save ALL changes to permanent memory';
	Xus_TN_INPUT_CONTROL.usa_TN_INPUT_CONTROL_DATA[14].in_Input_Option := INT#01;
	Xus_TN_INPUT_CONTROL.usa_TN_INPUT_CONTROL_DATA[14].in_Title_Y_Offset := INT#00;
	Xus_TN_INPUT_CONTROL.usa_TN_INPUT_CONTROL_DATA[14].in_Title_X_Offset := INT#00;
	Xus_TN_INPUT_CONTROL.usa_TN_INPUT_CONTROL_DATA[14].by_Title_Attr := BYTE#16#70;
	Xus_TN_INPUT_CONTROL.usa_TN_INPUT_CONTROL_DATA[14].st_Title_String := '';
	Xus_TN_INPUT_CONTROL.usa_TN_INPUT_CONTROL_DATA[14].st_Input_Mask := '    ';
	Xus_TN_INPUT_CONTROL.usa_TN_INPUT_CONTROL_DATA[14].st_Input_Data := 'SAVE';

	Xus_TN_INPUT_CONTROL.usa_TN_INPUT_CONTROL_DATA[15].in_Type := INT#02;
	Xus_TN_INPUT_CONTROL.usa_TN_INPUT_CONTROL_DATA[15].in_Y := INT#22;
	Xus_TN_INPUT_CONTROL.usa_TN_INPUT_CONTROL_DATA[15].in_X := INT#11;
	Xus_TN_INPUT_CONTROL.usa_TN_INPUT_CONTROL_DATA[15].by_Attr_mF := BYTE#16#07;
	Xus_TN_INPUT_CONTROL.usa_TN_INPUT_CONTROL_DATA[15].by_Attr_oF := BYTE#16#70;
	Xus_TN_INPUT_CONTROL.usa_TN_INPUT_CONTROL_DATA[15].st_Input_ToolTip := 'Apply changes';
	Xus_TN_INPUT_CONTROL.usa_TN_INPUT_CONTROL_DATA[15].in_Input_Option := INT#01;
	Xus_TN_INPUT_CONTROL.usa_TN_INPUT_CONTROL_DATA[15].in_Title_Y_Offset := INT#00;
	Xus_TN_INPUT_CONTROL.usa_TN_INPUT_CONTROL_DATA[15].in_Title_X_Offset := INT#00;
	Xus_TN_INPUT_CONTROL.usa_TN_INPUT_CONTROL_DATA[15].by_Title_Attr := BYTE#16#70;
	Xus_TN_INPUT_CONTROL.usa_TN_INPUT_CONTROL_DATA[15].st_Title_String := '';
	Xus_TN_INPUT_CONTROL.usa_TN_INPUT_CONTROL_DATA[15].st_Input_Mask := '     ';
	Xus_TN_INPUT_CONTROL.usa_TN_INPUT_CONTROL_DATA[15].st_Input_Data := 'APPLY';

	Xus_TN_INPUT_CONTROL.usa_TN_INPUT_CONTROL_DATA[16].in_Type := INT#02;
	Xus_TN_INPUT_CONTROL.usa_TN_INPUT_CONTROL_DATA[16].in_Y := INT#22;
	Xus_TN_INPUT_CONTROL.usa_TN_INPUT_CONTROL_DATA[16].in_X := INT#03;
	Xus_TN_INPUT_CONTROL.usa_TN_INPUT_CONTROL_DATA[16].by_Attr_mF := BYTE#16#07;
	Xus_TN_INPUT_CONTROL.usa_TN_INPUT_CONTROL_DATA[16].by_Attr_oF := BYTE#16#70;
	Xus_TN_INPUT_CONTROL.usa_TN_INPUT_CONTROL_DATA[16].st_Input_ToolTip := 'Return to Main Menu';
	Xus_TN_INPUT_CONTROL.usa_TN_INPUT_CONTROL_DATA[16].in_Input_Option := INT#01;
	Xus_TN_INPUT_CONTROL.usa_TN_INPUT_CONTROL_DATA[16].in_Title_Y_Offset := INT#00;
	Xus_TN_INPUT_CONTROL.usa_TN_INPUT_CONTROL_DATA[16].in_Title_X_Offset := INT#00;
	Xus_TN_INPUT_CONTROL.usa_TN_INPUT_CONTROL_DATA[16].by_Title_Attr := BYTE#16#70;
	Xus_TN_INPUT_CONTROL.usa_TN_INPUT_CONTROL_DATA[16].st_Title_String := '';
	Xus_TN_INPUT_CONTROL.usa_TN_INPUT_CONTROL_DATA[16].st_Input_Mask := '      ';
	Xus_TN_INPUT_CONTROL.usa_TN_INPUT_CONTROL_DATA[16].st_Input_Data := 'LOGOUT';

	(* Control-Tool-Tip *)
	Xus_TN_INPUT_CONTROL.in_ToolTip_Y := INT#23;
	Xus_TN_INPUT_CONTROL.in_ToolTip_X := INT#00;
	Xus_TN_INPUT_CONTROL.by_ToolTip_Attr := BYTE#07;
	Xus_TN_INPUT_CONTROL.in_ToolTip_Size := INT#80;

	(* Control-Verwaltung initialisieren *)
	Xus_TN_INPUT_CONTROL.in_Count := INT#16;
	Xus_TN_INPUT_CONTROL.bo_Enable := TRUE;
	Xus_TN_INPUT_CONTROL.bo_Reset_Fokus := TRUE;

END_IF;

IF (Xus_TN_SCREEN.in_Page_Number = INT#05) THEN

	(* eingegebenen String übernehmen *)
	IF Xus_TN_INPUT_CONTROL.usa_TN_INPUT_CONTROL_DATA[16].bo_Input_Entered = TRUE THEN

		Xus_TN_INPUT_CONTROL.usa_TN_INPUT_CONTROL_DATA[16].bo_Input_Entered := FALSE;
		Xus_TN_SCREEN.in_Page_Number := INT#00;
	END_IF;
END_IF;
END_PROGRAM

(* POU WORLD_WEATHER_DEMO, CFC *)
PROGRAM WORLD_WEATHER_DEMO
VAR
	IP_C: IP_C;
	S_BUF: NETWORK_BUFFER;
	R_BUF: NETWORK_BUFFER;
	IP_CONTROL_1: IP_CONTROL;
	activate: BOOL := TRUE;
	done: BOOL;
	busy: BOOL;
	error_c: DWORD;
	error_t: BYTE;
	latitude: REAL := 48.21;
	longitude: REAL := 16.37;
	WORLD_WEATHER: WORLD_WEATHER;
	WW_DATA: WORLD_WEATHER_DATA;
	CLK_PRG: CLK_PRG;
	WORLD_WEATHER_DESC_GE: WORLD_WEATHER_DESC_GE;
	WORLD_WEATHER_ICON_OSCAT: WORLD_WEATHER_ICON_OSCAT;
END_VAR
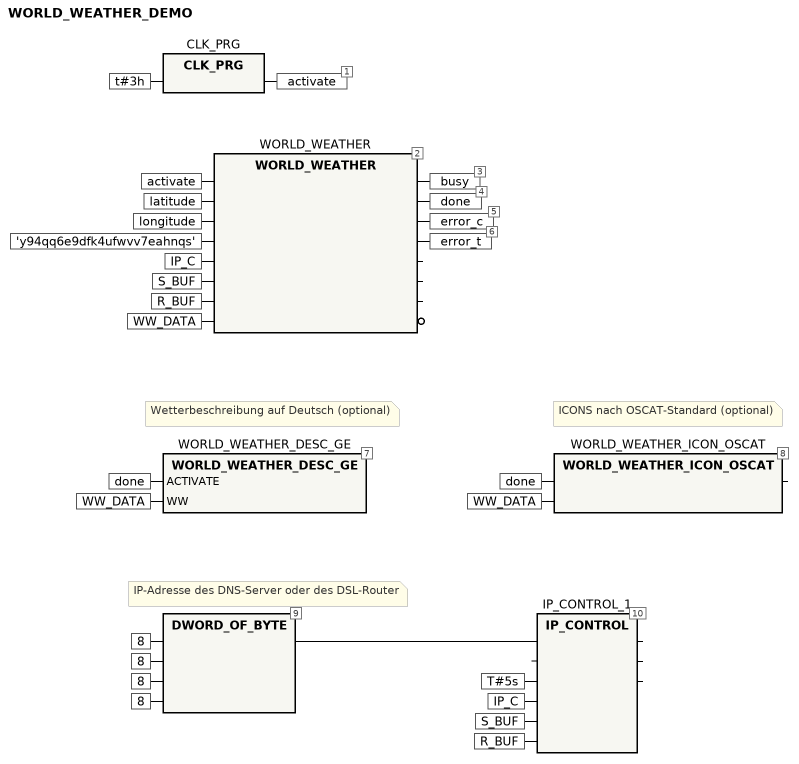
_CFC_ (* Continuous Function Chart, elements in execution order *)
#0 CLK_PRG:CLK_PRG(t#3h)
#1 activate <= #0
#2 WORLD_WEATHER:WORLD_WEATHER(activate, latitude, longitude, 'y94qq6e9dfk4ufwvv7eahnqs', IP_C, S_BUF, R_BUF, WW_DATA)
#3 busy <= #2.out 1
#4 done <= #2.out 2
#5 error_c <= #2.out 3
#6 error_t <= #2.out 4
#7 WORLD_WEATHER_DESC_GE:WORLD_WEATHER_DESC_GE(ACTIVATE: done, WW: WW_DATA)
#8 WORLD_WEATHER_ICON_OSCAT:WORLD_WEATHER_ICON_OSCAT(done, WW_DATA)
#9 DWORD_OF_BYTE(8, 8, 8, 8)
#10 IP_CONTROL_1:IP_CONTROL(#9, -, T#5s, IP_C, S_BUF, R_BUF)
(* ICONS nach OSCAT-Standard (optional) *)
(* IP-Adresse des DNS-Server oder des DSL-Router *)
(* Wetterbeschreibung auf Deutsch (optional) *)
_END_CFC_
END_PROGRAM

(* POU WORLD_WEATHER, ST *)
FUNCTION_BLOCK WORLD_WEATHER
VAR_IN_OUT
	IP_C : IP_C; (* IP_Control Verwaltungsstruktur *)
	S_BUF : NETWORK_BUFFER;
	R_BUF : NETWORK_BUFFER;
	WW : WORLD_WEATHER_DATA;
END_VAR
VAR_INPUT
	ACTIVATE : BOOL;
	LATITUDE : REAL;
	LONGITUDE : REAL;
	KEY : STRING(30);
END_VAR
VAR_OUTPUT
	BUSY : BOOL;
	DONE : BOOL;
	ERROR_C : DWORD;
	ERROR_T : BYTE;
END_VAR
VAR
	URL_DATA : url;
	DNS_CLIENT : DNS_CLIENT;
	HTTP_GET : HTTP_GET;
	CPB : CSV_PARSER_BUF;
	last_state : BOOL;
	value_int : INT;
	value_real : REAL;
	v_real : REAL;
	state : INT;
	url_str : STRING(STRING_LENGTH);
	offset : UDINT;
	size : INT;
	sep : BYTE;
	cnt : INT;
	day : INT;
	idx : INT;
	run : BYTE;
	result : BYTE;
	value : STRING(STRING_LENGTH);
	pos : INT;
END_VAR

(*

version 1.5	11. may 2013
programmer 	ks
tested by	ks

WORLD_WEATHER lädt von worldweather.com eine Wetter csv-datei und analysiert die Daten und legt diese in einem Array ab
Die Wetterdaten werden für 5 tage aufbereitet

*)
CASE state OF

00:
	IF ACTIVATE AND NOT last_state THEN
		state := 20;
		DONE := FALSE;
		BUSY := TRUE;
		ERROR_C := DWORD#0;
		ERROR_T := BYTE#0;
	END_IF;

20: (* URL for DNS UND HTTP-GET *)
	(* Example: http://api.worldweatheronline.com/free/v1/weather.ashx?q=48.21,16.37&format=csv&num_of_days=5&key=xxxxxxxxxxxxxxxxxxxxxx *)
	url_str := CONCAT('http://api.worldweatheronline.com/free/v1/weather.ashx?q=',REAL_TO_STRF(LATITUDE,6,D:='.'));
	url_str := CONCAT(url_str,',');
	url_str := CONCAT(url_str,REAL_TO_STRF(LONGITUDE,6,D:='.'));
	url_str := CONCAT(url_str,'&format=csv&num_of_days=5&key=');
	url_str := CONCAT(url_str,key);

	URL_DATA:=STRING_TO_URL(STR:=url_str, DEFAULT_PROTOCOL:='', DEFAULT_PATH:='' );
	state := 40;

40:
	IF DNS_CLIENT.DONE THEN
		state := 60;
	ELSIF (DNS_CLIENT.ERROR > DWORD#00) THEN
		(* Fehlerbehandlung *)
		ERROR_C := DNS_CLIENT.ERROR;
	ERROR_T := BYTE#01;
		state   := 100;
	END_IF;

60:
	IF HTTP_GET.DONE THEN
		sep := 0;
		idx := 0;
		day := 0;
		cnt := 0;
		OFFSET := HTTP_GET.BODY_START; (* Start Offset vorgeben *)
		size := HTTP_GET.BODY_STOP; (* End Position *)
		run := 1; (* Element suchen *)
		state := 80;

	ELSIF (HTTP_GET.ERROR > DWORD#00) THEN
		(* Fehlerbehandlung *)
		ERROR_C := HTTP_GET.ERROR;
		ERROR_T := BYTE#02;
		state := 100;
	END_IF;

80:	IF run = 0 THEN (* kein Befehl mehr aktiv ? *)
		run := 1; (*  nächstes Element suchen  *)
		IF result = 1 OR result = 2 THEN
			value_int := 0;
			value_real := 0.0;
			(* automatische konvertierung in real und int ausführen *)
			IF LEN(value) <= 20 THEN
				v_real:=FLOAT_TO_REAL(FLT:=value);
				IF CHK_REAL(v_real) = 0 THEN (* !!! prüft auf gültigen REAL Wert, ansonsten stürzt Twincat ab !!!!  *)
					value_real := v_real;
					value_int := REAL_TO_INT(value_real);
				END_IF;
			END_IF;
			cnt := cnt + 1;


			IF cnt = 1 AND LEFT(value,1) <> '#' THEN
				cnt := 0;
			END_IF;

